LIN {X 0,Y 573.917,Z 349.97,A -85,B 0,C 180,E1 -2263.779,E2 -2263.779} C_VEL
LIN {X 0,Y 573.417,Z 346.271,A -85,B 0,C 180,E1 -2263.85,E2 -2263.85} C_VEL
LIN {X 0,Y 573.634,Z 323.251,A -85,B 0,C 180,E1 -2266.915,E2 -2266.915} C_VEL
LIN {X 0,Y 573.847,Z 301.546,A -85,B 0,C 180,E1 -2269.849,E2 -2269.849} C_VEL
LIN {X 0,Y 574.055,Z 282.107,A -85,B 0,C 180,E1 -2272.493,E2 -2272.493} C_VEL
LIN {X 0,Y 574.049,Z 273.401,A -85,B 0,C 180,E1 -2273.681,E2 -2273.681} C_VEL
LIN {X 0,Y 573.25,Z 269.082,A -85,B 0,C 180,E1 -2274.344,E2 -2274.344} C_VEL
LIN {X 0,Y 573.182,Z 269.086,A -85,B 0,C 180,E1 -2276.978,E2 -2276.978} C_VEL
LIN {X 0,Y 573.215,Z 269.077,A -85,B 0,C 180,E1 -2279.482,E2 -2279.482} C_VEL
LIN {X 0,Y 573.242,Z 269.078,A -85,B 0,C 180,E1 -2282.226,E2 -2282.226} C_VEL
LIN {X 0,Y 573.214,Z 269.085,A -85,B 0,C 180,E1 -2284.768,E2 -2284.768} C_VEL
LIN {X 0,Y 573.204,Z 269.079,A -85,B 0,C 180,E1 -2287.807,E2 -2287.807} C_VEL
LIN {X 0,Y 573.23,Z 269.083,A -85,B 0,C 180,E1 -2290.523,E2 -2290.523} C_VEL
LIN {X 0,Y 573.189,Z 269.081,A -85,B 0,C 180,E1 -2293.36,E2 -2293.36} C_VEL
LIN {X 0,Y 573.213,Z 269.082,A -85,B 0,C 180,E1 -2296.33,E2 -2296.33} C_VEL
LIN {X 0,Y 573.222,Z 269.077,A -85,B 0,C 180,E1 -2299.473,E2 -2299.473} C_VEL
LIN {X 0,Y 573.201,Z 269.082,A -85,B 0,C 180,E1 -2302.189,E2 -2302.189} C_VEL
LIN {X 0,Y 573.199,Z 269.081,A -85,B 0,C 180,E1 -2305.228,E2 -2305.228} C_VEL
LIN {X 0,Y 573.21,Z 269.08,A -85,B 0,C 180,E1 -2308.182,E2 -2308.182} C_VEL
LIN {X 0,Y 573.206,Z 269.087,A -85,B 0,C 180,E1 -2310.631,E2 -2310.631} C_VEL
LIN {X 0,Y 573.178,Z 269.087,A -85,B 0,C 180,E1 -2313.02,E2 -2313.02} C_VEL
LIN {X 0,Y 573.181,Z 269.083,A -85,B 0,C 180,E1 -2315.361,E2 -2315.361} C_VEL
LIN {X 0,Y 573.185,Z 269.081,A -85,B 0,C 180,E1 -2317.66,E2 -2317.66} C_VEL
LIN {X 0,Y 573.227,Z 269.085,A -85,B 0,C 180,E1 -2320.668,E2 -2320.668} C_VEL
LIN {X 0,Y 573.205,Z 269.079,A -85,B 0,C 180,E1 -2323.62,E2 -2323.62} C_VEL
LIN {X 0,Y 573.192,Z 269.087,A -85,B 0,C 180,E1 -2326.528,E2 -2326.528} C_VEL
LIN {X 0,Y 573.243,Z 269.075,A -85,B 0,C 180,E1 -2329.403,E2 -2329.403} C_VEL
LIN {X 0,Y 573.241,Z 269.077,A -85,B 0,C 180,E1 -2332.249,E2 -2332.249} C_VEL
LIN {X 0,Y 573.271,Z 269.076,A -85,B 0,C 180,E1 -2335.077,E2 -2335.077} C_VEL
LIN {X 0,Y 573.256,Z 269.072,A -85,B 0,C 180,E1 -2337.892,E2 -2337.892} C_VEL
LIN {X 0,Y 573.307,Z 269.075,A -85,B 0,C 180,E1 -2340.702,E2 -2340.702} C_VEL
LIN {X 0,Y 573.204,Z 269.08,A -85,B 0,C 180,E1 -2343.514,E2 -2343.514} C_VEL
LIN {X 0,Y 573.254,Z 269.073,A -85,B 0,C 180,E1 -2345.628,E2 -2345.628} C_VEL
LIN {X 0,Y 573.267,Z 269.075,A -85,B 0,C 180,E1 -2348.459,E2 -2348.459} C_VEL
LIN {X 0,Y 573.284,Z 269.072,A -85,B 0,C 180,E1 -2351.311,E2 -2351.311} C_VEL
LIN {X 0,Y 573.239,Z 269.078,A -85,B 0,C 180,E1 -2354.425,E2 -2354.425} C_VEL
LIN {X 0,Y 573.221,Z 269.083,A -85,B 0,C 180,E1 -2357.112,E2 -2357.112} C_VEL
LIN {X 0,Y 573.224,Z 269.077,A -85,B 0,C 180,E1 -2360.077,E2 -2360.077} C_VEL
LIN {X 0,Y 573.206,Z 269.081,A -85,B 0,C 180,E1 -2362.339,E2 -2362.339} C_VEL
LIN {X 0,Y 573.216,Z 269.081,A -85,B 0,C 180,E1 -2364.415,E2 -2364.415} C_VEL
LIN {X 0,Y 572.592,Z 269.165,A -85,B 0,C 180,E1 -2365.001,E2 -2365.001} C_VEL
LIN {X 0,Y 569.754,Z 269.52,A -85,B 0,C 180,E1 -2365.953,E2 -2365.953} C_VEL
LIN {X 0,Y 567.326,Z 269.819,A -85,B 0,C 180,E1 -2366.719,E2 -2366.719} C_VEL
LIN {X 0,Y 566.274,Z 269.946,A -85,B 0,C 180,E1 -2367.31,E2 -2367.31} C_VEL
LIN {X 0,Y 566.184,Z 269.955,A -85,B 0,C 180,E1 -2367.511,E2 -2367.511} C_VEL
LIN {X 0,Y 566.163,Z 269.961,A -85,B 0,C 180,E1 -2370.593,E2 -2370.593} C_VEL
LIN {X 0,Y 566.198,Z 269.959,A -85,B 0,C 180,E1 -2373.103,E2 -2373.103} C_VEL
LIN {X 0,Y 566.185,Z 269.954,A -85,B 0,C 180,E1 -2375.69,E2 -2375.69} C_VEL
LIN {X 0,Y 566.191,Z 269.957,A -85,B 0,C 180,E1 -2378.561,E2 -2378.561} C_VEL
LIN {X 0,Y 566.196,Z 269.959,A -85,B 0,C 180,E1 -2381.137,E2 -2381.137} C_VEL
LIN {X 0,Y 566.177,Z 269.954,A -85,B 0,C 180,E1 -2384.037,E2 -2384.037} C_VEL
LIN {X 0,Y 566.19,Z 269.961,A -85,B 0,C 180,E1 -2387.084,E2 -2387.084} C_VEL
LIN {X 0,Y 566.209,Z 269.951,A -85,B 0,C 180,E1 -2389.805,E2 -2389.805} C_VEL
LIN {X 0,Y 566.183,Z 269.958,A -85,B 0,C 180,E1 -2392.601,E2 -2392.601} C_VEL
LIN {X 0,Y 566.205,Z 269.958,A -85,B 0,C 180,E1 -2395.185,E2 -2395.185} C_VEL
LIN {X 0,Y 566.222,Z 269.949,A -85,B 0,C 180,E1 -2397.745,E2 -2397.745} C_VEL
LIN {X 0,Y 566.193,Z 269.954,A -85,B 0,C 180,E1 -2400.329,E2 -2400.329} C_VEL
LIN {X 0,Y 566.21,Z 269.955,A -85,B 0,C 180,E1 -2402.663,E2 -2402.663} C_VEL
LIN {X 0,Y 566.229,Z 269.957,A -85,B 0,C 180,E1 -2405.04,E2 -2405.04} C_VEL
LIN {X 0,Y 566.187,Z 269.953,A -85,B 0,C 180,E1 -2408.138,E2 -2408.138} C_VEL
LIN {X 0,Y 566.231,Z 269.951,A -85,B 0,C 180,E1 -2410.613,E2 -2410.613} C_VEL
LIN {X 0,Y 566.212,Z 269.954,A -85,B 0,C 180,E1 -2413.413,E2 -2413.413} C_VEL
LIN {X 0,Y 566.193,Z 269.953,A -85,B 0,C 180,E1 -2416.359,E2 -2416.359} C_VEL
LIN {X 0,Y 566.232,Z 269.951,A -85,B 0,C 180,E1 -2418.675,E2 -2418.675} C_VEL
LIN {X 0,Y 566.23,Z 269.952,A -85,B 0,C 180,E1 -2421.434,E2 -2421.434} C_VEL
LIN {X 0,Y 566.255,Z 269.945,A -85,B 0,C 180,E1 -2424.301,E2 -2424.301} C_VEL
LIN {X 0,Y 566.282,Z 269.941,A -85,B 0,C 180,E1 -2427.865,E2 -2427.865} C_VEL
LIN {X 0,Y 566.297,Z 269.943,A -85,B 0,C 180,E1 -2430.71,E2 -2430.71} C_VEL
LIN {X 0,Y 566.268,Z 269.949,A -85,B 0,C 180,E1 -2432.844,E2 -2432.844} C_VEL
LIN {X 0,Y 566.261,Z 269.945,A -85,B 0,C 180,E1 -2435.697,E2 -2435.697} C_VEL
LIN {X 0,Y 566.224,Z 269.95,A -85,B 0,C 180,E1 -2438.564,E2 -2438.564} C_VEL
LIN {X 0,Y 566.235,Z 269.952,A -85,B 0,C 180,E1 -2441.452,E2 -2441.452} C_VEL
LIN {X 0,Y 566.226,Z 269.949,A -85,B 0,C 180,E1 -2444.505,E2 -2444.505} C_VEL
LIN {X 0,Y 566.194,Z 269.959,A -85,B 0,C 180,E1 -2447.329,E2 -2447.329} C_VEL
LIN {X 0,Y 566.209,Z 269.95,A -85,B 0,C 180,E1 -2450.334,E2 -2450.334} C_VEL
LIN {X 0,Y 566.216,Z 269.955,A -85,B 0,C 180,E1 -2453.399,E2 -2453.399} C_VEL
LIN {X 0,Y 566.21,Z 269.952,A -85,B 0,C 180,E1 -2455.745,E2 -2455.745} C_VEL
LIN {X 0,Y 566.19,Z 269.952,A -85,B 0,C 180,E1 -2458.2,E2 -2458.2} C_VEL
LIN {X 0,Y 566.185,Z 269.961,A -85,B 0,C 180,E1 -2461.076,E2 -2461.076} C_VEL
LIN {X 0,Y 566.205,Z 269.952,A -85,B 0,C 180,E1 -2463.734,E2 -2463.734} C_VEL
LIN {X 0,Y 566.191,Z 269.953,A -85,B 0,C 180,E1 -2466.565,E2 -2466.565} C_VEL
LIN {X 0,Y 566.188,Z 269.956,A -85,B 0,C 180,E1 -2469.683,E2 -2469.683} C_VEL
LIN {X 0,Y 566.197,Z 269.953,A -85,B 0,C 180,E1 -2472.082,E2 -2472.082} C_VEL
LIN {X 0,Y 566.254,Z 270.033,A -85,B 0,C 180,E1 -2474.364,E2 -2474.364} C_VEL
LIN {X 0,Y 566.279,Z 279.677,A -85,B 0,C 180,E1 -2476.263,E2 -2476.263} C_VEL
LIN {X 0,Y 566.19,Z 288.982,A -85,B 0,C 180,E1 -2478.061,E2 -2478.061} C_VEL
LIN {X 0,Y 567.187,Z 296.049,A -85,B 0,C 180,E1 -2478.176,E2 -2478.176} C_VEL
LIN {X 0,Y 566.936,Z 395.368,A -85,B 0,C 180,E1 -2479.456,E2 -2479.456} C_VEL
LIN {X 0,Y 566.826,Z 409.344,A -85,B 0,C 180,E1 -2479.796,E2 -2479.796} C_VEL
LIN {X 0,Y 566.705,Z 421.629,A -85,B 0,C 180,E1 -2480.246,E2 -2480.246} C_VEL
LIN {X 0,Y 566.564,Z 432.139,A -85,B 0,C 180,E1 -2480.756,E2 -2480.756} C_VEL
LIN {X 0,Y 566.42,Z 442.775,A -85,B 0,C 180,E1 -2481.406,E2 -2481.406} C_VEL
LIN {X 0,Y 566.365,Z 452.067,A -85,B 0,C 180,E1 -2482.104,E2 -2482.104} C_VEL
LIN {X 0,Y 566.234,Z 460.736,A -85,B 0,C 180,E1 -2482.886,E2 -2482.886} C_VEL
LIN {X 0,Y 566.136,Z 469.017,A -85,B 0,C 180,E1 -2483.785,E2 -2483.785} C_VEL
LIN {X 0,Y 566.01,Z 477.294,A -85,B 0,C 180,E1 -2484.886,E2 -2484.886} C_VEL
LIN {X 0,Y 565.945,Z 484.05,A -85,B 0,C 180,E1 -2486.026,E2 -2486.026} C_VEL
LIN {X 0,Y 565.918,Z 488.182,A -85,B 0,C 180,E1 -2486.878,E2 -2486.878} C_VEL
LIN {X 0,Y 565.884,Z 492.888,A -85,B 0,C 180,E1 -2488.142,E2 -2488.142} C_VEL
LIN {X 0,Y 565.877,Z 496.169,A -85,B 0,C 180,E1 -2489.39,E2 -2489.39} C_VEL
LIN {X 0,Y 565.861,Z 497.855,A -85,B 0,C 180,E1 -2490.377,E2 -2490.377} C_VEL
LIN {X 0,Y 565.838,Z 498.588,A -85,B 0,C 180,E1 -2491.027,E2 -2491.027} C_VEL
LIN {X 0,Y 565.818,Z 498.965,A -85,B 0,C 180,E1 -2491.858,E2 -2491.858} C_VEL
LIN {X 0,Y 565.834,Z 498.805,A -85,B 0,C 180,E1 -2492.642,E2 -2492.642} C_VEL
LIN {X 0,Y 565.85,Z 498.2,A -85,B 0,C 180,E1 -2493.441,E2 -2493.441} C_VEL
LIN {X 0,Y 565.858,Z 497.121,A -85,B 0,C 180,E1 -2494.234,E2 -2494.234} C_VEL
LIN {X 0,Y 565.897,Z 494.476,A -85,B 0,C 180,E1 -2495.419,E2 -2495.419} C_VEL
LIN {X 0,Y 565.928,Z 490.68,A -85,B 0,C 180,E1 -2496.585,E2 -2496.585} C_VEL
LIN {X 0,Y 565.95,Z 485.642,A -85,B 0,C 180,E1 -2497.744,E2 -2497.744} C_VEL
LIN {X 0,Y 565.99,Z 480.913,A -85,B 0,C 180,E1 -2498.619,E2 -2498.619} C_VEL
LIN {X 0,Y 566.094,Z 474.044,A -85,B 0,C 180,E1 -2499.659,E2 -2499.659} C_VEL
LIN {X 0,Y 566.157,Z 466.342,A -85,B 0,C 180,E1 -2500.615,E2 -2500.615} C_VEL
LIN {X 0,Y 566.322,Z 456.139,A -85,B 0,C 180,E1 -2501.646,E2 -2501.646} C_VEL
LIN {X 0,Y 566.385,Z 445.594,A -85,B 0,C 180,E1 -2502.488,E2 -2502.488} C_VEL
LIN {X 0,Y 566.539,Z 436.194,A -85,B 0,C 180,E1 -2503.101,E2 -2503.101} C_VEL
LIN {X 0,Y 566.628,Z 426.691,A -85,B 0,C 180,E1 -2503.61,E2 -2503.61} C_VEL
LIN {X 0,Y 566.755,Z 416.899,A -85,B 0,C 180,E1 -2504.03,E2 -2504.03} C_VEL
LIN {X 0,Y 566.837,Z 406.261,A -85,B 0,C 180,E1 -2504.379,E2 -2504.379} C_VEL
LIN {X 0,Y 566.92,Z 394.133,A -85,B 0,C 180,E1 -2504.658,E2 -2504.658} C_VEL
LIN {X 0,Y 567.05,Z 293.787,A -85,B 0,C 180,E1 -2505.946,E2 -2505.946} C_VEL
LIN {X 0,Y 566.183,Z 288.859,A -85,B 0,C 180,E1 -2506.038,E2 -2506.038} C_VEL
LIN {X 0,Y 566.336,Z 273.977,A -85,B 0,C 180,E1 -2508.945,E2 -2508.945} C_VEL
LIN {X 0,Y 566.174,Z 269.958,A -85,B 0,C 180,E1 -2509.767,E2 -2509.767} C_VEL
LIN {X 0,Y 566.183,Z 269.955,A -85,B 0,C 180,E1 -2512.153,E2 -2512.153} C_VEL
LIN {X 0,Y 566.23,Z 269.957,A -85,B 0,C 180,E1 -2515.016,E2 -2515.016} C_VEL
LIN {X 0,Y 566.211,Z 269.951,A -85,B 0,C 180,E1 -2517.866,E2 -2517.866} C_VEL
LIN {X 0,Y 566.256,Z 269.951,A -85,B 0,C 180,E1 -2520.711,E2 -2520.711} C_VEL
LIN {X 0,Y 566.146,Z 269.96,A -85,B 0,C 180,E1 -2523.559,E2 -2523.559} C_VEL
LIN {X 0,Y 566.208,Z 269.951,A -85,B 0,C 180,E1 -2525.699,E2 -2525.699} C_VEL
LIN {X 0,Y 566.192,Z 269.956,A -85,B 0,C 180,E1 -2528.567,E2 -2528.567} C_VEL
LIN {X 0,Y 566.203,Z 269.954,A -85,B 0,C 180,E1 -2531.455,E2 -2531.455} C_VEL
LIN {X 0,Y 566.173,Z 269.957,A -85,B 0,C 180,E1 -2534.509,E2 -2534.509} C_VEL
LIN {X 0,Y 566.149,Z 269.962,A -85,B 0,C 180,E1 -2537.334,E2 -2537.334} C_VEL
LIN {X 0,Y 566.158,Z 269.958,A -85,B 0,C 180,E1 -2539.583,E2 -2539.583} C_VEL
LIN {X 0,Y 566.144,Z 269.958,A -85,B 0,C 180,E1 -2541.865,E2 -2541.865} C_VEL
LIN {X 0,Y 566.181,Z 269.962,A -85,B 0,C 180,E1 -2545.037,E2 -2545.037} C_VEL
LIN {X 0,Y 566.179,Z 269.96,A -85,B 0,C 180,E1 -2547.341,E2 -2547.341} C_VEL
LIN {X 0,Y 566.153,Z 269.958,A -85,B 0,C 180,E1 -2549.772,E2 -2549.772} C_VEL
LIN {X 0,Y 566.161,Z 269.956,A -85,B 0,C 180,E1 -2552.434,E2 -2552.434} C_VEL
LIN {X 0,Y 566.168,Z 269.961,A -85,B 0,C 180,E1 -2554.998,E2 -2554.998} C_VEL
LIN {X 0,Y 566.155,Z 269.962,A -85,B 0,C 180,E1 -2557.464,E2 -2557.464} C_VEL
LIN {X 0,Y 566.188,Z 269.952,A -85,B 0,C 180,E1 -2560.201,E2 -2560.201} C_VEL
LIN {X 0,Y 566.168,Z 269.961,A -85,B 0,C 180,E1 -2563.058,E2 -2563.058} C_VEL
LIN {X 0,Y 566.166,Z 269.956,A -85,B 0,C 180,E1 -2566.053,E2 -2566.053} C_VEL
LIN {X 0,Y 566.179,Z 269.957,A -85,B 0,C 180,E1 -2568.867,E2 -2568.867} C_VEL
LIN {X 0,Y 566.158,Z 269.961,A -85,B 0,C 180,E1 -2571.641,E2 -2571.641} C_VEL
LIN {X 0,Y 566.139,Z 269.959,A -85,B 0,C 180,E1 -2574.312,E2 -2574.312} C_VEL
LIN {X 0,Y 566.186,Z 269.958,A -85,B 0,C 180,E1 -2576.901,E2 -2576.901} C_VEL
LIN {X 0,Y 566.162,Z 269.967,A -85,B 0,C 180,E1 -2579.411,E2 -2579.411} C_VEL
LIN {X 0,Y 566.172,Z 269.959,A -85,B 0,C 180,E1 -2581.86,E2 -2581.86} C_VEL
LIN {X 0,Y 566.191,Z 269.955,A -85,B 0,C 180,E1 -2584.254,E2 -2584.254} C_VEL
LIN {X 0,Y 566.235,Z 270.017,A -85,B 0,C 180,E1 -2585.703,E2 -2585.703} C_VEL
LIN {X 0,Y 567.056,Z 275.86,A -85,B 0,C 180,E1 -2586.513,E2 -2586.513} C_VEL
LIN {X 0,Y 566.955,Z 296.913,A -85,B 0,C 180,E1 -2589.315,E2 -2589.315} C_VEL
LIN {X 0,Y 566.727,Z 315.073,A -85,B 0,C 180,E1 -2591.755,E2 -2591.755} C_VEL
LIN {X 0,Y 566.527,Z 334.178,A -85,B 0,C 180,E1 -2594.349,E2 -2594.349} C_VEL
LIN {X 0,Y 566.431,Z 346.452,A -85,B 0,C 180,E1 -2595.99,E2 -2595.99} C_VEL
LIN {X 0,Y 567.179,Z 352.712,A -85,B 0,C 180,E1 -2596.089,E2 -2596.089} C_VEL
LIN {X 0,Y 566.977,Z 455.07,A -85,B 0,C 180,E1 -2597.406,E2 -2597.406} C_VEL
LIN {X 0,Y 566.845,Z 467.537,A -85,B 0,C 180,E1 -2597.698,E2 -2597.698} C_VEL
LIN {X 0,Y 566.722,Z 480.435,A -85,B 0,C 180,E1 -2598.15,E2 -2598.15} C_VEL
LIN {X 0,Y 566.63,Z 492.077,A -85,B 0,C 180,E1 -2598.704,E2 -2598.704} C_VEL
LIN {X 0,Y 566.474,Z 502.939,A -85,B 0,C 180,E1 -2599.367,E2 -2599.367} C_VEL
LIN {X 0,Y 566.332,Z 513.565,A -85,B 0,C 180,E1 -2600.178,E2 -2600.178} C_VEL
LIN {X 0,Y 566.206,Z 523.133,A -85,B 0,C 180,E1 -2601.076,E2 -2601.076} C_VEL
LIN {X 0,Y 566.111,Z 530.976,A -85,B 0,C 180,E1 -2601.974,E2 -2601.974} C_VEL
LIN {X 0,Y 566,Z 538.634,A -85,B 0,C 180,E1 -2603.048,E2 -2603.048} C_VEL
LIN {X 0,Y 566.003,Z 545.688,A -85,B 0,C 180,E1 -2604.301,E2 -2604.301} C_VEL
LIN {X 0,Y 565.933,Z 550.379,A -85,B 0,C 180,E1 -2605.372,E2 -2605.372} C_VEL
LIN {X 0,Y 565.926,Z 553.962,A -85,B 0,C 180,E1 -2606.442,E2 -2606.442} C_VEL
LIN {X 0,Y 565.878,Z 555.811,A -85,B 0,C 180,E1 -2607.154,E2 -2607.154} C_VEL
LIN {X 0,Y 565.845,Z 558.186,A -85,B 0,C 180,E1 -2608.578,E2 -2608.578} C_VEL
LIN {X 0,Y 565.839,Z 559,A -85,B 0,C 180,E1 -2610.001,E2 -2610.001} C_VEL
LIN {X 0,Y 565.845,Z 558.185,A -85,B 0,C 180,E1 -2611.424,E2 -2611.424} C_VEL
LIN {X 0,Y 565.878,Z 555.808,A -85,B 0,C 180,E1 -2612.848,E2 -2612.848} C_VEL
LIN {X 0,Y 565.927,Z 552.893,A -85,B 0,C 180,E1 -2613.917,E2 -2613.917} C_VEL
LIN {X 0,Y 565.878,Z 548.946,A -85,B 0,C 180,E1 -2614.988,E2 -2614.988} C_VEL
LIN {X 0,Y 566.002,Z 543.864,A -85,B 0,C 180,E1 -2616.059,E2 -2616.059} C_VEL
LIN {X 0,Y 566.041,Z 537.465,A -85,B 0,C 180,E1 -2617.133,E2 -2617.133} C_VEL
LIN {X 0,Y 566.134,Z 529.475,A -85,B 0,C 180,E1 -2618.208,E2 -2618.208} C_VEL
LIN {X 0,Y 566.229,Z 521.333,A -85,B 0,C 180,E1 -2619.106,E2 -2619.106} C_VEL
LIN {X 0,Y 566.342,Z 511.398,A -85,B 0,C 180,E1 -2620.005,E2 -2620.005} C_VEL
LIN {X 0,Y 566.529,Z 500.301,A -85,B 0,C 180,E1 -2620.807,E2 -2620.807} C_VEL
LIN {X 0,Y 566.641,Z 489.175,A -85,B 0,C 180,E1 -2621.446,E2 -2621.446} C_VEL
LIN {X 0,Y 566.741,Z 476.983,A -85,B 0,C 180,E1 -2621.988,E2 -2621.988} C_VEL
LIN {X 0,Y 566.864,Z 464.18,A -85,B 0,C 180,E1 -2622.394,E2 -2622.394} C_VEL
LIN {X 0,Y 566.979,Z 450.61,A -85,B 0,C 180,E1 -2622.665,E2 -2622.665} C_VEL
LIN {X 0,Y 567.031,Z 350.74,A -85,B 0,C 180,E1 -2623.94,E2 -2623.94} C_VEL
LIN {X 0,Y 566.441,Z 346.271,A -85,B 0,C 180,E1 -2624.024,E2 -2624.024} C_VEL
LIN {X 0,Y 566.694,Z 322.246,A -85,B 0,C 180,E1 -2627.265,E2 -2627.265} C_VEL
LIN {X 0,Y 566.952,Z 299.903,A -85,B 0,C 180,E1 -2630.309,E2 -2630.309} C_VEL
LIN {X 0,Y 567.192,Z 279,A -85,B 0,C 180,E1 -2633.166,E2 -2633.166} C_VEL
LIN {X 0,Y 566.866,Z 273.321,A -85,B 0,C 180,E1 -2633.968,E2 -2633.968} C_VEL
LIN {X 0,Y 566.192,Z 269.962,A -85,B 0,C 180,E1 -2634.472,E2 -2634.472} C_VEL
LIN {X 0,Y 566.16,Z 269.958,A -85,B 0,C 180,E1 -2637.34,E2 -2637.34} C_VEL
LIN {X 0,Y 566.163,Z 269.956,A -85,B 0,C 180,E1 -2639.769,E2 -2639.769} C_VEL
LIN {X 0,Y 566.194,Z 269.959,A -85,B 0,C 180,E1 -2642.428,E2 -2642.428} C_VEL
LIN {X 0,Y 566.158,Z 269.96,A -85,B 0,C 180,E1 -2644.986,E2 -2644.986} C_VEL
LIN {X 0,Y 566.172,Z 269.955,A -85,B 0,C 180,E1 -2647.46,E2 -2647.46} C_VEL
LIN {X 0,Y 566.19,Z 269.955,A -85,B 0,C 180,E1 -2650.197,E2 -2650.197} C_VEL
LIN {X 0,Y 566.169,Z 269.959,A -85,B 0,C 180,E1 -2653.053,E2 -2653.053} C_VEL
LIN {X 0,Y 566.154,Z 269.958,A -85,B 0,C 180,E1 -2656.049,E2 -2656.049} C_VEL
LIN {X 0,Y 566.179,Z 269.956,A -85,B 0,C 180,E1 -2659.213,E2 -2659.213} C_VEL
LIN {X 0,Y 566.152,Z 269.957,A -85,B 0,C 180,E1 -2661.634,E2 -2661.634} C_VEL
LIN {X 0,Y 566.12,Z 269.965,A -85,B 0,C 180,E1 -2664.304,E2 -2664.304} C_VEL
LIN {X 0,Y 566.168,Z 269.962,A -85,B 0,C 180,E1 -2666.894,E2 -2666.894} C_VEL
LIN {X 0,Y 566.141,Z 269.959,A -85,B 0,C 180,E1 -2669.404,E2 -2669.404} C_VEL
LIN {X 0,Y 566.158,Z 269.957,A -85,B 0,C 180,E1 -2671.854,E2 -2671.854} C_VEL
LIN {X 0,Y 566.157,Z 269.96,A -85,B 0,C 180,E1 -2674.248,E2 -2674.248} C_VEL
LIN {X 0,Y 566.133,Z 269.961,A -85,B 0,C 180,E1 -2677.366,E2 -2677.366} C_VEL
LIN {X 0,Y 566.165,Z 269.956,A -85,B 0,C 180,E1 -2679.661,E2 -2679.661} C_VEL
LIN {X 0,Y 566.159,Z 269.965,A -85,B 0,C 180,E1 -2682.667,E2 -2682.667} C_VEL
LIN {X 0,Y 566.173,Z 269.955,A -85,B 0,C 180,E1 -2685.625,E2 -2685.625} C_VEL
LIN {X 0,Y 566.237,Z 269.955,A -85,B 0,C 180,E1 -2688.652,E2 -2688.652} C_VEL
LIN {X 0,Y 566.183,Z 269.955,A -85,B 0,C 180,E1 -2691.433,E2 -2691.433} C_VEL
LIN {X 0,Y 566.223,Z 269.951,A -85,B 0,C 180,E1 -2694.301,E2 -2694.301} C_VEL
LIN {X 0,Y 566.228,Z 269.948,A -85,B 0,C 180,E1 -2697.866,E2 -2697.866} C_VEL
LIN {X 0,Y 566.276,Z 269.95,A -85,B 0,C 180,E1 -2700.711,E2 -2700.711} C_VEL
LIN {X 0,Y 566.155,Z 269.958,A -85,B 0,C 180,E1 -2703.558,E2 -2703.558} C_VEL
LIN {X 0,Y 566.221,Z 269.949,A -85,B 0,C 180,E1 -2705.698,E2 -2705.698} C_VEL
LIN {X 0,Y 566.209,Z 269.956,A -85,B 0,C 180,E1 -2708.566,E2 -2708.566} C_VEL
LIN {X 0,Y 566.223,Z 269.95,A -85,B 0,C 180,E1 -2711.454,E2 -2711.454} C_VEL
LIN {X 0,Y 566.192,Z 269.957,A -85,B 0,C 180,E1 -2714.507,E2 -2714.507} C_VEL
LIN {X 0,Y 566.167,Z 269.959,A -85,B 0,C 180,E1 -2717.332,E2 -2717.332} C_VEL
LIN {X 0,Y 566.177,Z 269.955,A -85,B 0,C 180,E1 -2719.581,E2 -2719.581} C_VEL
LIN {X 0,Y 566.162,Z 269.956,A -85,B 0,C 180,E1 -2721.863,E2 -2721.863} C_VEL
LIN {X 0,Y 566.181,Z 269.962,A -85,B 0,C 180,E1 -2725.031,E2 -2725.031} C_VEL
LIN {X 0,Y 566.184,Z 269.955,A -85,B 0,C 180,E1 -2727.511,E2 -2727.511} C_VEL
LIN {X 0,Y 565.506,Z 270.039,A -85,B 0,C 180,E1 -2728.105,E2 -2728.105} C_VEL
LIN {X 0,Y 562.64,Z 270.402,A -85,B 0,C 180,E1 -2729.068,E2 -2729.068} C_VEL
LIN {X 0,Y 560.23,Z 270.699,A -85,B 0,C 180,E1 -2729.844,E2 -2729.844} C_VEL
LIN {X 0,Y 559.202,Z 270.827,A -85,B 0,C 180,E1 -2730.443,E2 -2730.443} C_VEL
LIN {X 0,Y 559.122,Z 270.837,A -85,B 0,C 180,E1 -2730.645,E2 -2730.645} C_VEL
LIN {X 0,Y 559.147,Z 270.831,A -85,B 0,C 180,E1 -2733.575,E2 -2733.575} C_VEL
LIN {X 0,Y 559.162,Z 270.831,A -85,B 0,C 180,E1 -2736.453,E2 -2736.453} C_VEL
LIN {X 0,Y 559.153,Z 270.838,A -85,B 0,C 180,E1 -2738.935,E2 -2738.935} C_VEL
LIN {X 0,Y 559.174,Z 270.827,A -85,B 0,C 180,E1 -2741.769,E2 -2741.769} C_VEL
LIN {X 0,Y 559.117,Z 270.841,A -85,B 0,C 180,E1 -2744.741,E2 -2744.741} C_VEL
LIN {X 0,Y 559.149,Z 270.835,A -85,B 0,C 180,E1 -2747.259,E2 -2747.259} C_VEL
LIN {X 0,Y 559.169,Z 270.828,A -85,B 0,C 180,E1 -2750.137,E2 -2750.137} C_VEL
LIN {X 0,Y 559.132,Z 270.841,A -85,B 0,C 180,E1 -2752.894,E2 -2752.894} C_VEL
LIN {X 0,Y 559.141,Z 270.833,A -85,B 0,C 180,E1 -2755.557,E2 -2755.557} C_VEL
LIN {X 0,Y 559.157,Z 270.829,A -85,B 0,C 180,E1 -2758.139,E2 -2758.139} C_VEL
LIN {X 0,Y 559.134,Z 270.836,A -85,B 0,C 180,E1 -2760.648,E2 -2760.648} C_VEL
LIN {X 0,Y 559.163,Z 270.836,A -85,B 0,C 180,E1 -2763.173,E2 -2763.173} C_VEL
LIN {X 0,Y 559.149,Z 270.833,A -85,B 0,C 180,E1 -2765.496,E2 -2765.496} C_VEL
LIN {X 0,Y 559.165,Z 270.832,A -85,B 0,C 180,E1 -2768.625,E2 -2768.625} C_VEL
LIN {X 0,Y 559.164,Z 270.837,A -85,B 0,C 180,E1 -2770.927,E2 -2770.927} C_VEL
LIN {X 0,Y 559.163,Z 270.828,A -85,B 0,C 180,E1 -2773.948,E2 -2773.948} C_VEL
LIN {X 0,Y 559.168,Z 270.828,A -85,B 0,C 180,E1 -2776.184,E2 -2776.184} C_VEL
LIN {X 0,Y 559.193,Z 270.833,A -85,B 0,C 180,E1 -2779.133,E2 -2779.133} C_VEL
LIN {X 0,Y 559.203,Z 270.823,A -85,B 0,C 180,E1 -2782.053,E2 -2782.053} C_VEL
LIN {X 0,Y 559.25,Z 270.825,A -85,B 0,C 180,E1 -2784.953,E2 -2784.953} C_VEL
LIN {X 0,Y 559.253,Z 270.817,A -85,B 0,C 180,E1 -2787.838,E2 -2787.838} C_VEL
LIN {X 0,Y 559.268,Z 270.819,A -85,B 0,C 180,E1 -2790.719,E2 -2790.719} C_VEL
LIN {X 0,Y 559.235,Z 270.825,A -85,B 0,C 180,E1 -2792.88,E2 -2792.88} C_VEL
LIN {X 0,Y 559.229,Z 270.821,A -85,B 0,C 180,E1 -2795.768,E2 -2795.768} C_VEL
LIN {X 0,Y 559.183,Z 270.829,A -85,B 0,C 180,E1 -2798.672,E2 -2798.672} C_VEL
LIN {X 0,Y 559.199,Z 270.826,A -85,B 0,C 180,E1 -2801.598,E2 -2801.598} C_VEL
LIN {X 0,Y 559.191,Z 270.826,A -85,B 0,C 180,E1 -2804.593,E2 -2804.593} C_VEL
LIN {X 0,Y 559.154,Z 270.833,A -85,B 0,C 180,E1 -2807.554,E2 -2807.554} C_VEL
LIN {X 0,Y 559.164,Z 270.829,A -85,B 0,C 180,E1 -2809.834,E2 -2809.834} C_VEL
LIN {X 0,Y 559.143,Z 270.83,A -85,B 0,C 180,E1 -2812.149,E2 -2812.149} C_VEL
LIN {X 0,Y 559.145,Z 270.831,A -85,B 0,C 180,E1 -2814.502,E2 -2814.502} C_VEL
LIN {X 0,Y 559.165,Z 270.833,A -85,B 0,C 180,E1 -2816.898,E2 -2816.898} C_VEL
LIN {X 0,Y 559.169,Z 270.828,A -85,B 0,C 180,E1 -2819.862,E2 -2819.862} C_VEL
LIN {X 0,Y 559.154,Z 270.831,A -85,B 0,C 180,E1 -2822.71,E2 -2822.71} C_VEL
LIN {X 0,Y 559.135,Z 270.839,A -85,B 0,C 180,E1 -2825.318,E2 -2825.318} C_VEL
LIN {X 0,Y 559.109,Z 270.834,A -85,B 0,C 180,E1 -2828.013,E2 -2828.013} C_VEL
LIN {X 0,Y 559.148,Z 270.834,A -85,B 0,C 180,E1 -2830.807,E2 -2830.807} C_VEL
LIN {X 0,Y 559.162,Z 270.835,A -85,B 0,C 180,E1 -2833.725,E2 -2833.725} C_VEL
LIN {X 0,Y 559.25,Z 271.036,A -85,B 0,C 180,E1 -2834.347,E2 -2834.347} C_VEL
LIN {X 0,Y 559.215,Z 282.244,A -85,B 0,C 180,E1 -2836.566,E2 -2836.566} C_VEL
LIN {X 0,Y 559.142,Z 288.907,A -85,B 0,C 180,E1 -2837.88,E2 -2837.88} C_VEL
LIN {X 0,Y 560.301,Z 296.457,A -85,B 0,C 180,E1 -2838.008,E2 -2838.008} C_VEL
LIN {X 0,Y 560.02,Z 395.757,A -85,B 0,C 180,E1 -2839.306,E2 -2839.306} C_VEL
LIN {X 0,Y 559.904,Z 409.255,A -85,B 0,C 180,E1 -2839.64,E2 -2839.64} C_VEL
LIN {X 0,Y 559.744,Z 421.917,A -85,B 0,C 180,E1 -2840.111,E2 -2840.111} C_VEL
LIN {X 0,Y 559.584,Z 432.524,A -85,B 0,C 180,E1 -2840.636,E2 -2840.636} C_VEL
LIN {X 0,Y 559.446,Z 441.889,A -85,B 0,C 180,E1 -2841.211,E2 -2841.211} C_VEL
LIN {X 0,Y 559.325,Z 450.942,A -85,B 0,C 180,E1 -2841.884,E2 -2841.884} C_VEL
LIN {X 0,Y 559.209,Z 458.95,A -85,B 0,C 180,E1 -2842.593,E2 -2842.593} C_VEL
LIN {X 0,Y 559.118,Z 467.038,A -85,B 0,C 180,E1 -2843.449,E2 -2843.449} C_VEL
LIN {X 0,Y 559.017,Z 473.256,A -85,B 0,C 180,E1 -2844.226,E2 -2844.226} C_VEL
LIN {X 0,Y 558.933,Z 479.627,A -85,B 0,C 180,E1 -2845.174,E2 -2845.174} C_VEL
LIN {X 0,Y 558.857,Z 484.722,A -85,B 0,C 180,E1 -2846.087,E2 -2846.087} C_VEL
LIN {X 0,Y 558.848,Z 488.275,A -85,B 0,C 180,E1 -2846.836,E2 -2846.836} C_VEL
LIN {X 0,Y 558.813,Z 492.949,A -85,B 0,C 180,E1 -2848.115,E2 -2848.115} C_VEL
LIN {X 0,Y 558.771,Z 495.323,A -85,B 0,C 180,E1 -2848.957,E2 -2848.957} C_VEL
LIN {X 0,Y 558.755,Z 497.653,A -85,B 0,C 180,E1 -2850.201,E2 -2850.201} C_VEL
LIN {X 0,Y 558.731,Z 498.899,A -85,B 0,C 180,E1 -2851.689,E2 -2851.689} C_VEL
LIN {X 0,Y 558.73,Z 498.588,A -85,B 0,C 180,E1 -2853.075,E2 -2853.075} C_VEL
LIN {X 0,Y 558.743,Z 497.661,A -85,B 0,C 180,E1 -2853.881,E2 -2853.881} C_VEL
LIN {X 0,Y 558.76,Z 495.832,A -85,B 0,C 180,E1 -2854.89,E2 -2854.89} C_VEL
LIN {X 0,Y 558.822,Z 493.245,A -85,B 0,C 180,E1 -2855.875,E2 -2855.875} C_VEL
LIN {X 0,Y 558.843,Z 489.063,A -85,B 0,C 180,E1 -2857.055,E2 -2857.055} C_VEL
LIN {X 0,Y 558.889,Z 483.723,A -85,B 0,C 180,E1 -2858.205,E2 -2858.205} C_VEL
LIN {X 0,Y 558.967,Z 476.663,A -85,B 0,C 180,E1 -2859.388,E2 -2859.388} C_VEL
LIN {X 0,Y 559.078,Z 469.121,A -85,B 0,C 180,E1 -2860.396,E2 -2860.396} C_VEL
LIN {X 0,Y 559.2,Z 460.847,A -85,B 0,C 180,E1 -2861.308,E2 -2861.308} C_VEL
LIN {X 0,Y 559.295,Z 452.57,A -85,B 0,C 180,E1 -2862.07,E2 -2862.07} C_VEL
LIN {X 0,Y 559.387,Z 444.539,A -85,B 0,C 180,E1 -2862.694,E2 -2862.694} C_VEL
LIN {X 0,Y 559.6,Z 435.068,A -85,B 0,C 180,E1 -2863.305,E2 -2863.305} C_VEL
LIN {X 0,Y 559.677,Z 426.249,A -85,B 0,C 180,E1 -2863.776,E2 -2863.776} C_VEL
LIN {X 0,Y 559.77,Z 416.393,A -85,B 0,C 180,E1 -2864.2,E2 -2864.2} C_VEL
LIN {X 0,Y 559.892,Z 405.519,A -85,B 0,C 180,E1 -2864.553,E2 -2864.553} C_VEL
LIN {X 0,Y 560.015,Z 393.606,A -85,B 0,C 180,E1 -2864.824,E2 -2864.824} C_VEL
LIN {X 0,Y 560.185,Z 294.859,A -85,B 0,C 180,E1 -2866.106,E2 -2866.106} C_VEL
LIN {X 0,Y 559.152,Z 288.797,A -85,B 0,C 180,E1 -2866.23,E2 -2866.23} C_VEL
LIN {X 0,Y 559.221,Z 276.702,A -85,B 0,C 180,E1 -2868.563,E2 -2868.563} C_VEL
LIN {X 0,Y 559.177,Z 270.831,A -85,B 0,C 180,E1 -2869.637,E2 -2869.637} C_VEL
LIN {X 0,Y 559.142,Z 270.84,A -85,B 0,C 180,E1 -2872.78,E2 -2872.78} C_VEL
LIN {X 0,Y 559.203,Z 270.833,A -85,B 0,C 180,E1 -2874.953,E2 -2874.953} C_VEL
LIN {X 0,Y 559.184,Z 270.826,A -85,B 0,C 180,E1 -2877.84,E2 -2877.84} C_VEL
LIN {X 0,Y 559.224,Z 270.827,A -85,B 0,C 180,E1 -2880.72,E2 -2880.72} C_VEL
LIN {X 0,Y 559.191,Z 270.833,A -85,B 0,C 180,E1 -2882.882,E2 -2882.882} C_VEL
LIN {X 0,Y 559.175,Z 270.827,A -85,B 0,C 180,E1 -2885.771,E2 -2885.771} C_VEL
LIN {X 0,Y 559.147,Z 270.835,A -85,B 0,C 180,E1 -2888.675,E2 -2888.675} C_VEL
LIN {X 0,Y 559.154,Z 270.831,A -85,B 0,C 180,E1 -2891.602,E2 -2891.602} C_VEL
LIN {X 0,Y 559.139,Z 270.834,A -85,B 0,C 180,E1 -2894.598,E2 -2894.598} C_VEL
LIN {X 0,Y 559.109,Z 270.836,A -85,B 0,C 180,E1 -2897.559,E2 -2897.559} C_VEL
LIN {X 0,Y 559.12,Z 270.833,A -85,B 0,C 180,E1 -2899.84,E2 -2899.84} C_VEL
LIN {X 0,Y 559.09,Z 270.836,A -85,B 0,C 180,E1 -2902.155,E2 -2902.155} C_VEL
LIN {X 0,Y 559.132,Z 270.838,A -85,B 0,C 180,E1 -2905.301,E2 -2905.301} C_VEL
LIN {X 0,Y 559.146,Z 270.831,A -85,B 0,C 180,E1 -2907.714,E2 -2907.714} C_VEL
LIN {X 0,Y 559.117,Z 270.841,A -85,B 0,C 180,E1 -2911.022,E2 -2911.022} C_VEL
LIN {X 0,Y 559.132,Z 270.831,A -85,B 0,C 180,E1 -2913.955,E2 -2913.955} C_VEL
LIN {X 0,Y 559.104,Z 270.844,A -85,B 0,C 180,E1 -2917.112,E2 -2917.112} C_VEL
LIN {X 0,Y 559.131,Z 270.832,A -85,B 0,C 180,E1 -2919.947,E2 -2919.947} C_VEL
LIN {X 0,Y 559.128,Z 270.834,A -85,B 0,C 180,E1 -2922.747,E2 -2922.747} C_VEL
LIN {X 0,Y 559.12,Z 270.836,A -85,B 0,C 180,E1 -2925.765,E2 -2925.765} C_VEL
LIN {X 0,Y 559.158,Z 270.828,A -85,B 0,C 180,E1 -2928.236,E2 -2928.236} C_VEL
LIN {X 0,Y 559.147,Z 270.838,A -85,B 0,C 180,E1 -2931.196,E2 -2931.196} C_VEL
LIN {X 0,Y 559.115,Z 270.838,A -85,B 0,C 180,E1 -2933.793,E2 -2933.793} C_VEL
LIN {X 0,Y 559.138,Z 270.833,A -85,B 0,C 180,E1 -2936.429,E2 -2936.429} C_VEL
LIN {X 0,Y 559.136,Z 270.838,A -85,B 0,C 180,E1 -2938.984,E2 -2938.984} C_VEL
LIN {X 0,Y 559.153,Z 270.837,A -85,B 0,C 180,E1 -2941.623,E2 -2941.623} C_VEL
LIN {X 0,Y 559.162,Z 270.832,A -85,B 0,C 180,E1 -2944.705,E2 -2944.705} C_VEL
LIN {X 0,Y 559.216,Z 270.974,A -85,B 0,C 180,E1 -2945.6,E2 -2945.6} C_VEL
LIN {X 0,Y 560.099,Z 277.032,A -85,B 0,C 180,E1 -2946.459,E2 -2946.459} C_VEL
LIN {X 0,Y 559.934,Z 299.004,A -85,B 0,C 180,E1 -2949.428,E2 -2949.428} C_VEL
LIN {X 0,Y 559.729,Z 321.817,A -85,B 0,C 180,E1 -2952.465,E2 -2952.465} C_VEL
LIN {X 0,Y 559.443,Z 343.73,A -85,B 0,C 180,E1 -2955.451,E2 -2955.451} C_VEL
LIN {X 0,Y 559.435,Z 346.452,A -85,B 0,C 180,E1 -2955.811,E2 -2955.811} C_VEL
LIN {X 0,Y 560.293,Z 353.439,A -85,B 0,C 180,E1 -2955.924,E2 -2955.924} C_VEL
LIN {X 0,Y 560.052,Z 455.069,A -85,B 0,C 180,E1 -2957.248,E2 -2957.248} C_VEL
LIN {X 0,Y 559.925,Z 467.537,A -85,B 0,C 180,E1 -2957.544,E2 -2957.544} C_VEL
LIN {X 0,Y 559.761,Z 480.437,A -85,B 0,C 180,E1 -2958.001,E2 -2958.001} C_VEL
LIN {X 0,Y 559.665,Z 491.854,A -85,B 0,C 180,E1 -2958.549,E2 -2958.549} C_VEL
LIN {X 0,Y 559.491,Z 502.937,A -85,B 0,C 180,E1 -2959.233,E2 -2959.233} C_VEL
LIN {X 0,Y 559.311,Z 513.564,A -85,B 0,C 180,E1 -2960.053,E2 -2960.053} C_VEL
LIN {X 0,Y 559.16,Z 523.133,A -85,B 0,C 180,E1 -2960.963,E2 -2960.963} C_VEL
LIN {X 0,Y 559.048,Z 530.976,A -85,B 0,C 180,E1 -2961.872,E2 -2961.872} C_VEL
LIN {X 0,Y 558.941,Z 538.634,A -85,B 0,C 180,E1 -2962.96,E2 -2962.96} C_VEL
LIN {X 0,Y 558.935,Z 545.688,A -85,B 0,C 180,E1 -2964.229,E2 -2964.229} C_VEL
LIN {X 0,Y 558.826,Z 550.379,A -85,B 0,C 180,E1 -2965.313,E2 -2965.313} C_VEL
LIN {X 0,Y 558.836,Z 553.962,A -85,B 0,C 180,E1 -2966.396,E2 -2966.396} C_VEL
LIN {X 0,Y 558.799,Z 555.811,A -85,B 0,C 180,E1 -2967.118,E2 -2967.118} C_VEL
LIN {X 0,Y 558.745,Z 558.185,A -85,B 0,C 180,E1 -2968.56,E2 -2968.56} C_VEL
LIN {X 0,Y 558.74,Z 559,A -85,B 0,C 180,E1 -2970.001,E2 -2970.001} C_VEL
LIN {X 0,Y 558.745,Z 558.184,A -85,B 0,C 180,E1 -2971.443,E2 -2971.443} C_VEL
LIN {X 0,Y 558.799,Z 555.808,A -85,B 0,C 180,E1 -2972.885,E2 -2972.885} C_VEL
LIN {X 0,Y 558.844,Z 552.893,A -85,B 0,C 180,E1 -2973.967,E2 -2973.967} C_VEL
LIN {X 0,Y 558.798,Z 548.946,A -85,B 0,C 180,E1 -2975.051,E2 -2975.051} C_VEL
LIN {X 0,Y 558.922,Z 543.864,A -85,B 0,C 180,E1 -2976.136,E2 -2976.136} C_VEL
LIN {X 0,Y 558.978,Z 537.464,A -85,B 0,C 180,E1 -2977.223,E2 -2977.223} C_VEL
LIN {X 0,Y 559.099,Z 529.475,A -85,B 0,C 180,E1 -2978.312,E2 -2978.312} C_VEL
LIN {X 0,Y 559.185,Z 521.332,A -85,B 0,C 180,E1 -2979.221,E2 -2979.221} C_VEL
LIN {X 0,Y 559.343,Z 511.397,A -85,B 0,C 180,E1 -2980.132,E2 -2980.132} C_VEL
LIN {X 0,Y 559.535,Z 500.378,A -85,B 0,C 180,E1 -2980.938,E2 -2980.938} C_VEL
LIN {X 0,Y 559.672,Z 488.459,A -85,B 0,C 180,E1 -2981.628,E2 -2981.628} C_VEL
LIN {X 0,Y 559.809,Z 475.77,A -85,B 0,C 180,E1 -2982.185,E2 -2982.185} C_VEL
LIN {X 0,Y 559.966,Z 462.35,A -85,B 0,C 180,E1 -2982.596,E2 -2982.596} C_VEL
LIN {X 0,Y 560.062,Z 449.094,A -85,B 0,C 180,E1 -2982.847,E2 -2982.847} C_VEL
LIN {X 0,Y 560.237,Z 352.132,A -85,B 0,C 180,E1 -2984.095,E2 -2984.095} C_VEL
LIN {X 0,Y 559.427,Z 346.271,A -85,B 0,C 180,E1 -2984.203,E2 -2984.203} C_VEL
LIN {X 0,Y 559.709,Z 323.839,A -85,B 0,C 180,E1 -2987.264,E2 -2987.264} C_VEL
LIN {X 0,Y 559.992,Z 300.981,A -85,B 0,C 180,E1 -2990.38,E2 -2990.38} C_VEL
LIN {X 0,Y 560.264,Z 278.681,A -85,B 0,C 180,E1 -2993.469,E2 -2993.469} C_VEL
LIN {X 0,Y 559.901,Z 274.529,A -85,B 0,C 180,E1 -2994.074,E2 -2994.074} C_VEL
LIN {X 0,Y 559.159,Z 270.838,A -85,B 0,C 180,E1 -2994.649,E2 -2994.649} C_VEL
LIN {X 0,Y 559.109,Z 270.841,A -85,B 0,C 180,E1 -2996.904,E2 -2996.904} C_VEL
LIN {X 0,Y 559.11,Z 270.835,A -85,B 0,C 180,E1 -2999.354,E2 -2999.354} C_VEL
LIN {X 0,Y 559.156,Z 270.829,A -85,B 0,C 180,E1 -3001.861,E2 -3001.861} C_VEL
LIN {X 0,Y 559.121,Z 270.84,A -85,B 0,C 180,E1 -3004.444,E2 -3004.444} C_VEL
LIN {X 0,Y 559.112,Z 270.837,A -85,B 0,C 180,E1 -3007.108,E2 -3007.108} C_VEL
LIN {X 0,Y 559.142,Z 270.831,A -85,B 0,C 180,E1 -3009.939,E2 -3009.939} C_VEL
LIN {X 0,Y 559.132,Z 270.84,A -85,B 0,C 180,E1 -3012.742,E2 -3012.742} C_VEL
LIN {X 0,Y 559.114,Z 270.834,A -85,B 0,C 180,E1 -3015.761,E2 -3015.761} C_VEL
LIN {X 0,Y 559.104,Z 270.838,A -85,B 0,C 180,E1 -3018.224,E2 -3018.224} C_VEL
LIN {X 0,Y 559.145,Z 270.832,A -85,B 0,C 180,E1 -3021.19,E2 -3021.19} C_VEL
LIN {X 0,Y 559.093,Z 270.837,A -85,B 0,C 180,E1 -3023.785,E2 -3023.785} C_VEL
LIN {X 0,Y 559.116,Z 270.839,A -85,B 0,C 180,E1 -3026.422,E2 -3026.422} C_VEL
LIN {X 0,Y 559.122,Z 270.838,A -85,B 0,C 180,E1 -3028.978,E2 -3028.978} C_VEL
LIN {X 0,Y 559.111,Z 270.834,A -85,B 0,C 180,E1 -3031.621,E2 -3031.621} C_VEL
LIN {X 0,Y 559.125,Z 270.833,A -85,B 0,C 180,E1 -3033.9,E2 -3033.9} C_VEL
LIN {X 0,Y 559.078,Z 270.843,A -85,B 0,C 180,E1 -3037.064,E2 -3037.064} C_VEL
LIN {X 0,Y 559.135,Z 270.833,A -85,B 0,C 180,E1 -3039.393,E2 -3039.393} C_VEL
LIN {X 0,Y 559.099,Z 270.836,A -85,B 0,C 180,E1 -3041.684,E2 -3041.684} C_VEL
LIN {X 0,Y 559.125,Z 270.833,A -85,B 0,C 180,E1 -3043.946,E2 -3043.946} C_VEL
LIN {X 0,Y 559.123,Z 270.835,A -85,B 0,C 180,E1 -3046.183,E2 -3046.183} C_VEL
LIN {X 0,Y 559.198,Z 270.828,A -85,B 0,C 180,E1 -3049.133,E2 -3049.133} C_VEL
LIN {X 0,Y 559.163,Z 270.829,A -85,B 0,C 180,E1 -3052.053,E2 -3052.053} C_VEL
LIN {X 0,Y 559.217,Z 270.829,A -85,B 0,C 180,E1 -3054.953,E2 -3054.953} C_VEL
LIN {X 0,Y 559.201,Z 270.823,A -85,B 0,C 180,E1 -3057.839,E2 -3057.839} C_VEL
LIN {X 0,Y 559.244,Z 270.826,A -85,B 0,C 180,E1 -3060.72,E2 -3060.72} C_VEL
LIN {X 0,Y 559.208,Z 270.832,A -85,B 0,C 180,E1 -3062.881,E2 -3062.881} C_VEL
LIN {X 0,Y 559.189,Z 270.825,A -85,B 0,C 180,E1 -3065.77,E2 -3065.77} C_VEL
LIN {X 0,Y 559.165,Z 270.836,A -85,B 0,C 180,E1 -3068.674,E2 -3068.674} C_VEL
LIN {X 0,Y 559.174,Z 270.827,A -85,B 0,C 180,E1 -3071.601,E2 -3071.601} C_VEL
LIN {X 0,Y 559.159,Z 270.835,A -85,B 0,C 180,E1 -3074.596,E2 -3074.596} C_VEL
LIN {X 0,Y 559.127,Z 270.834,A -85,B 0,C 180,E1 -3077.558,E2 -3077.558} C_VEL
LIN {X 0,Y 559.151,Z 270.836,A -85,B 0,C 180,E1 -3080.605,E2 -3080.605} C_VEL
LIN {X 0,Y 559.11,Z 270.835,A -85,B 0,C 180,E1 -3083.718,E2 -3083.718} C_VEL
LIN {X 0,Y 559.166,Z 270.828,A -85,B 0,C 180,E1 -3086.097,E2 -3086.097} C_VEL
LIN {X 0,Y 559.133,Z 270.836,A -85,B 0,C 180,E1 -3088.531,E2 -3088.531} C_VEL
LIN {X 0,Y 559.122,Z 270.837,A -85,B 0,C 180,E1 -3090.645,E2 -3090.645} C_VEL
LIN {X 0,Y 558.46,Z 270.924,A -85,B 0,C 180,E1 -3091.247,E2 -3091.247} C_VEL
LIN {X 0,Y 555.597,Z 271.28,A -85,B 0,C 180,E1 -3092.223,E2 -3092.223} C_VEL
LIN {X 0,Y 553.185,Z 271.581,A -85,B 0,C 180,E1 -3093.009,E2 -3093.009} C_VEL
LIN {X 0,Y 552.167,Z 271.701,A -85,B 0,C 180,E1 -3093.616,E2 -3093.616} C_VEL
LIN {X 0,Y 552.095,Z 271.709,A -85,B 0,C 180,E1 -3093.821,E2 -3093.821} C_VEL
LIN {X 0,Y 552.09,Z 271.717,A -85,B 0,C 180,E1 -3096.748,E2 -3096.748} C_VEL
LIN {X 0,Y 552.109,Z 271.709,A -85,B 0,C 180,E1 -3099.528,E2 -3099.528} C_VEL
LIN {X 0,Y 552.107,Z 271.71,A -85,B 0,C 180,E1 -3102.427,E2 -3102.427} C_VEL
LIN {X 0,Y 552.078,Z 271.713,A -85,B 0,C 180,E1 -3105.565,E2 -3105.565} C_VEL
LIN {X 0,Y 552.126,Z 271.711,A -85,B 0,C 180,E1 -3108.677,E2 -3108.677} C_VEL
LIN {X 0,Y 552.104,Z 271.711,A -85,B 0,C 180,E1 -3111.413,E2 -3111.413} C_VEL
LIN {X 0,Y 552.099,Z 271.709,A -85,B 0,C 180,E1 -3114.16,E2 -3114.16} C_VEL
LIN {X 0,Y 552.099,Z 271.716,A -85,B 0,C 180,E1 -3116.815,E2 -3116.815} C_VEL
LIN {X 0,Y 552.094,Z 271.713,A -85,B 0,C 180,E1 -3119.392,E2 -3119.392} C_VEL
LIN {X 0,Y 552.117,Z 271.706,A -85,B 0,C 180,E1 -3121.904,E2 -3121.904} C_VEL
LIN {X 0,Y 552.147,Z 271.707,A -85,B 0,C 180,E1 -3124.651,E2 -3124.651} C_VEL
LIN {X 0,Y 552.086,Z 271.712,A -85,B 0,C 180,E1 -3127.55,E2 -3127.55} C_VEL
LIN {X 0,Y 552.144,Z 271.704,A -85,B 0,C 180,E1 -3130.374,E2 -3130.374} C_VEL
LIN {X 0,Y 552.151,Z 271.711,A -85,B 0,C 180,E1 -3132.978,E2 -3132.978} C_VEL
LIN {X 0,Y 552.132,Z 271.704,A -85,B 0,C 180,E1 -3136.005,E2 -3136.005} C_VEL
LIN {X 0,Y 552.16,Z 271.71,A -85,B 0,C 180,E1 -3138.993,E2 -3138.993} C_VEL
LIN {X 0,Y 552.157,Z 271.701,A -85,B 0,C 180,E1 -3141.951,E2 -3141.951} C_VEL
LIN {X 0,Y 552.225,Z 271.699,A -85,B 0,C 180,E1 -3144.888,E2 -3144.888} C_VEL
LIN {X 0,Y 552.224,Z 271.693,A -85,B 0,C 180,E1 -3147.811,E2 -3147.811} C_VEL
LIN {X 0,Y 552.239,Z 271.695,A -85,B 0,C 180,E1 -3150.728,E2 -3150.728} C_VEL
LIN {X 0,Y 552.202,Z 271.702,A -85,B 0,C 180,E1 -3152.917,E2 -3152.917} C_VEL
LIN {X 0,Y 552.198,Z 271.696,A -85,B 0,C 180,E1 -3155.842,E2 -3155.842} C_VEL
LIN {X 0,Y 552.154,Z 271.706,A -85,B 0,C 180,E1 -3158.784,E2 -3158.784} C_VEL
LIN {X 0,Y 552.156,Z 271.702,A -85,B 0,C 180,E1 -3161.748,E2 -3161.748} C_VEL
LIN {X 0,Y 552.129,Z 271.708,A -85,B 0,C 180,E1 -3164.746,E2 -3164.746} C_VEL
LIN {X 0,Y 552.105,Z 271.708,A -85,B 0,C 180,E1 -3167.786,E2 -3167.786} C_VEL
LIN {X 0,Y 552.123,Z 271.705,A -85,B 0,C 180,E1 -3170.098,E2 -3170.098} C_VEL
LIN {X 0,Y 552.101,Z 271.708,A -85,B 0,C 180,E1 -3172.447,E2 -3172.447} C_VEL
LIN {X 0,Y 552.14,Z 271.709,A -85,B 0,C 180,E1 -3175.348,E2 -3175.348} C_VEL
LIN {X 0,Y 552.11,Z 271.706,A -85,B 0,C 180,E1 -3178.094,E2 -3178.094} C_VEL
LIN {X 0,Y 552.095,Z 271.71,A -85,B 0,C 180,E1 -3180.605,E2 -3180.605} C_VEL
LIN {X 0,Y 552.106,Z 271.717,A -85,B 0,C 180,E1 -3183.181,E2 -3183.181} C_VEL
LIN {X 0,Y 552.088,Z 271.71,A -85,B 0,C 180,E1 -3185.838,E2 -3185.838} C_VEL
LIN {X 0,Y 552.099,Z 271.715,A -85,B 0,C 180,E1 -3189.059,E2 -3189.059} C_VEL
LIN {X 0,Y 552.139,Z 271.711,A -85,B 0,C 180,E1 -3191.438,E2 -3191.438} C_VEL
LIN {X 0,Y 552.165,Z 271.77,A -85,B 0,C 180,E1 -3194.265,E2 -3194.265} C_VEL
LIN {X 0,Y 552.236,Z 280.86,A -85,B 0,C 180,E1 -3196.074,E2 -3196.074} C_VEL
LIN {X 0,Y 552.144,Z 289.057,A -85,B 0,C 180,E1 -3197.692,E2 -3197.692} C_VEL
LIN {X 0,Y 553.395,Z 297.217,A -85,B 0,C 180,E1 -3197.838,E2 -3197.838} C_VEL
LIN {X 0,Y 553.122,Z 395.02,A -85,B 0,C 180,E1 -3199.129,E2 -3199.129} C_VEL
LIN {X 0,Y 552.986,Z 407.989,A -85,B 0,C 180,E1 -3199.447,E2 -3199.447} C_VEL
LIN {X 0,Y 552.802,Z 421.471,A -85,B 0,C 180,E1 -3199.939,E2 -3199.939} C_VEL
LIN {X 0,Y 552.605,Z 432.909,A -85,B 0,C 180,E1 -3200.514,E2 -3200.514} C_VEL
LIN {X 0,Y 552.471,Z 441.351,A -85,B 0,C 180,E1 -3201.035,E2 -3201.035} C_VEL
LIN {X 0,Y 552.31,Z 450.268,A -85,B 0,C 180,E1 -3201.697,E2 -3201.697} C_VEL
LIN {X 0,Y 552.201,Z 458.819,A -85,B 0,C 180,E1 -3202.46,E2 -3202.46} C_VEL
LIN {X 0,Y 552.074,Z 466.799,A -85,B 0,C 180,E1 -3203.312,E2 -3203.312} C_VEL
LIN {X 0,Y 551.971,Z 473.407,A -85,B 0,C 180,E1 -3204.148,E2 -3204.148} C_VEL
LIN {X 0,Y 551.844,Z 479.313,A -85,B 0,C 180,E1 -3205.034,E2 -3205.034} C_VEL
LIN {X 0,Y 551.804,Z 484.258,A -85,B 0,C 180,E1 -3205.917,E2 -3205.917} C_VEL
LIN {X 0,Y 551.776,Z 488.361,A -85,B 0,C 180,E1 -3206.792,E2 -3206.792} C_VEL
LIN {X 0,Y 551.747,Z 491.686,A -85,B 0,C 180,E1 -3207.658,E2 -3207.658} C_VEL
LIN {X 0,Y 551.706,Z 494.463,A -85,B 0,C 180,E1 -3208.582,E2 -3208.582} C_VEL
LIN {X 0,Y 551.671,Z 497.447,A -85,B 0,C 180,E1 -3210.017,E2 -3210.017} C_VEL
LIN {X 0,Y 551.629,Z 498.617,A -85,B 0,C 180,E1 -3211.045,E2 -3211.045} C_VEL
LIN {X 0,Y 551.645,Z 498.968,A -85,B 0,C 180,E1 -3211.876,E2 -3211.876} C_VEL
LIN {X 0,Y 551.631,Z 498.588,A -85,B 0,C 180,E1 -3213.09,E2 -3213.09} C_VEL
LIN {X 0,Y 551.667,Z 497.041,A -85,B 0,C 180,E1 -3214.333,E2 -3214.333} C_VEL
LIN {X 0,Y 551.717,Z 494.355,A -85,B 0,C 180,E1 -3215.544,E2 -3215.544} C_VEL
LIN {X 0,Y 551.748,Z 490.508,A -85,B 0,C 180,E1 -3216.743,E2 -3216.743} C_VEL
LIN {X 0,Y 551.797,Z 487.333,A -85,B 0,C 180,E1 -3217.537,E2 -3217.537} C_VEL
LIN {X 0,Y 551.839,Z 481.162,A -85,B 0,C 180,E1 -3218.742,E2 -3218.742} C_VEL
LIN {X 0,Y 551.953,Z 475.129,A -85,B 0,C 180,E1 -3219.698,E2 -3219.698} C_VEL
LIN {X 0,Y 552.027,Z 469.323,A -85,B 0,C 180,E1 -3220.478,E2 -3220.478} C_VEL
LIN {X 0,Y 552.125,Z 462.577,A -85,B 0,C 180,E1 -3221.252,E2 -3221.252} C_VEL
LIN {X 0,Y 552.285,Z 453.455,A -85,B 0,C 180,E1 -3222.122,E2 -3222.122} C_VEL
LIN {X 0,Y 552.39,Z 445.322,A -85,B 0,C 180,E1 -3222.773,E2 -3222.773} C_VEL
LIN {X 0,Y 552.606,Z 436.349,A -85,B 0,C 180,E1 -3223.373,E2 -3223.373} C_VEL
LIN {X 0,Y 552.719,Z 426.81,A -85,B 0,C 180,E1 -3223.898,E2 -3223.898} C_VEL
LIN {X 0,Y 552.841,Z 417.08,A -85,B 0,C 180,E1 -3224.328,E2 -3224.328} C_VEL
LIN {X 0,Y 552.971,Z 406.753,A -85,B 0,C 180,E1 -3224.677,E2 -3224.677} C_VEL
LIN {X 0,Y 553.081,Z 394.963,A -85,B 0,C 180,E1 -3224.963,E2 -3224.963} C_VEL
LIN {X 0,Y 553.348,Z 295.929,A -85,B 0,C 180,E1 -3226.27,E2 -3226.27} C_VEL
LIN {X 0,Y 552.134,Z 288.968,A -85,B 0,C 180,E1 -3226.404,E2 -3226.404} C_VEL
LIN {X 0,Y 552.172,Z 275.63,A -85,B 0,C 180,E1 -3228.819,E2 -3228.819} C_VEL
LIN {X 0,Y 552.107,Z 271.713,A -85,B 0,C 180,E1 -3229.457,E2 -3229.457} C_VEL
LIN {X 0,Y 552.104,Z 271.709,A -85,B 0,C 180,E1 -3231.951,E2 -3231.951} C_VEL
LIN {X 0,Y 552.176,Z 271.709,A -85,B 0,C 180,E1 -3234.889,E2 -3234.889} C_VEL
LIN {X 0,Y 552.156,Z 271.702,A -85,B 0,C 180,E1 -3237.812,E2 -3237.812} C_VEL
LIN {X 0,Y 552.193,Z 271.703,A -85,B 0,C 180,E1 -3240.73,E2 -3240.73} C_VEL
LIN {X 0,Y 552.157,Z 271.71,A -85,B 0,C 180,E1 -3242.919,E2 -3242.919} C_VEL
LIN {X 0,Y 552.143,Z 271.703,A -85,B 0,C 180,E1 -3245.845,E2 -3245.845} C_VEL
LIN {X 0,Y 552.115,Z 271.712,A -85,B 0,C 180,E1 -3248.787,E2 -3248.787} C_VEL
LIN {X 0,Y 552.107,Z 271.707,A -85,B 0,C 180,E1 -3251.752,E2 -3251.752} C_VEL
LIN {X 0,Y 552.079,Z 271.716,A -85,B 0,C 180,E1 -3254.75,E2 -3254.75} C_VEL
LIN {X 0,Y 552.061,Z 271.712,A -85,B 0,C 180,E1 -3257.79,E2 -3257.79} C_VEL
LIN {X 0,Y 552.079,Z 271.709,A -85,B 0,C 180,E1 -3260.104,E2 -3260.104} C_VEL
LIN {X 0,Y 552.043,Z 271.716,A -85,B 0,C 180,E1 -3262.453,E2 -3262.453} C_VEL
LIN {X 0,Y 552.11,Z 271.711,A -85,B 0,C 180,E1 -3265.355,E2 -3265.355} C_VEL
LIN {X 0,Y 552.077,Z 271.71,A -85,B 0,C 180,E1 -3268.1,E2 -3268.1} C_VEL
LIN {X 0,Y 552.06,Z 271.715,A -85,B 0,C 180,E1 -3270.612,E2 -3270.612} C_VEL
LIN {X 0,Y 552.083,Z 271.719,A -85,B 0,C 180,E1 -3273.188,E2 -3273.188} C_VEL
LIN {X 0,Y 552.065,Z 271.713,A -85,B 0,C 180,E1 -3275.846,E2 -3275.846} C_VEL
LIN {X 0,Y 552.087,Z 271.717,A -85,B 0,C 180,E1 -3279.066,E2 -3279.066} C_VEL
LIN {X 0,Y 552.134,Z 271.709,A -85,B 0,C 180,E1 -3281.445,E2 -3281.445} C_VEL
LIN {X 0,Y 552.06,Z 271.713,A -85,B 0,C 180,E1 -3284.536,E2 -3284.536} C_VEL
LIN {X 0,Y 552.101,Z 271.713,A -85,B 0,C 180,E1 -3287.588,E2 -3287.588} C_VEL
LIN {X 0,Y 552.103,Z 271.708,A -85,B 0,C 180,E1 -3290.477,E2 -3290.477} C_VEL
LIN {X 0,Y 552.082,Z 271.72,A -85,B 0,C 180,E1 -3293.321,E2 -3293.321} C_VEL
LIN {X 0,Y 552.105,Z 271.711,A -85,B 0,C 180,E1 -3295.943,E2 -3295.943} C_VEL
LIN {X 0,Y 552.101,Z 271.711,A -85,B 0,C 180,E1 -3298.544,E2 -3298.544} C_VEL
LIN {X 0,Y 552.108,Z 271.716,A -85,B 0,C 180,E1 -3301.442,E2 -3301.442} C_VEL
LIN {X 0,Y 552.113,Z 271.709,A -85,B 0,C 180,E1 -3304.359,E2 -3304.359} C_VEL
LIN {X 0,Y 552.166,Z 271.826,A -85,B 0,C 180,E1 -3305.494,E2 -3305.494} C_VEL
LIN {X 0,Y 553.144,Z 278.866,A -85,B 0,C 180,E1 -3306.477,E2 -3306.477} C_VEL
LIN {X 0,Y 552.908,Z 301.204,A -85,B 0,C 180,E1 -3309.543,E2 -3309.543} C_VEL
LIN {X 0,Y 552.662,Z 323.088,A -85,B 0,C 180,E1 -3312.506,E2 -3312.506} C_VEL
LIN {X 0,Y 552.433,Z 345.08,A -85,B 0,C 180,E1 -3315.451,E2 -3315.451} C_VEL
LIN {X 0,Y 552.447,Z 346.442,A -85,B 0,C 180,E1 -3315.628,E2 -3315.628} C_VEL
LIN {X 0,Y 553.389,Z 354.507,A -85,B 0,C 180,E1 -3315.758,E2 -3315.758} C_VEL
LIN {X 0,Y 553.137,Z 455.069,A -85,B 0,C 180,E1 -3317.085,E2 -3317.085} C_VEL
LIN {X 0,Y 552.991,Z 467.536,A -85,B 0,C 180,E1 -3317.385,E2 -3317.385} C_VEL
LIN {X 0,Y 552.85,Z 479.976,A -85,B 0,C 180,E1 -3317.829,E2 -3317.829} C_VEL
LIN {X 0,Y 552.68,Z 491.855,A -85,B 0,C 180,E1 -3318.403,E2 -3318.403} C_VEL
LIN {X 0,Y 552.493,Z 502.935,A -85,B 0,C 180,E1 -3319.095,E2 -3319.095} C_VEL
LIN {X 0,Y 552.29,Z 513.562,A -85,B 0,C 180,E1 -3319.925,E2 -3319.925} C_VEL
LIN {X 0,Y 552.124,Z 523.133,A -85,B 0,C 180,E1 -3320.847,E2 -3320.847} C_VEL
LIN {X 0,Y 552.012,Z 530.976,A -85,B 0,C 180,E1 -3321.767,E2 -3321.767} C_VEL
LIN {X 0,Y 551.887,Z 538.633,A -85,B 0,C 180,E1 -3322.87,E2 -3322.87} C_VEL
LIN {X 0,Y 551.866,Z 545.688,A -85,B 0,C 180,E1 -3324.154,E2 -3324.154} C_VEL
LIN {X 0,Y 551.725,Z 550.379,A -85,B 0,C 180,E1 -3325.252,E2 -3325.252} C_VEL
LIN {X 0,Y 551.75,Z 553.963,A -85,B 0,C 180,E1 -3326.35,E2 -3326.35} C_VEL
LIN {X 0,Y 551.723,Z 555.81,A -85,B 0,C 180,E1 -3327.081,E2 -3327.081} C_VEL
LIN {X 0,Y 551.645,Z 558.184,A -85,B 0,C 180,E1 -3328.541,E2 -3328.541} C_VEL
LIN {X 0,Y 551.64,Z 559,A -85,B 0,C 180,E1 -3330.001,E2 -3330.001} C_VEL
LIN {X 0,Y 551.645,Z 558.183,A -85,B 0,C 180,E1 -3331.461,E2 -3331.461} C_VEL
LIN {X 0,Y 551.724,Z 555.808,A -85,B 0,C 180,E1 -3332.922,E2 -3332.922} C_VEL
LIN {X 0,Y 551.764,Z 552.893,A -85,B 0,C 180,E1 -3334.018,E2 -3334.018} C_VEL
LIN {X 0,Y 551.724,Z 548.946,A -85,B 0,C 180,E1 -3335.116,E2 -3335.116} C_VEL
LIN {X 0,Y 551.803,Z 543.189,A -85,B 0,C 180,E1 -3336.341,E2 -3336.341} C_VEL
LIN {X 0,Y 551.927,Z 536.233,A -85,B 0,C 180,E1 -3337.5,E2 -3337.5} C_VEL
LIN {X 0,Y 552.083,Z 527.989,A -85,B 0,C 180,E1 -3338.603,E2 -3338.603} C_VEL
LIN {X 0,Y 552.224,Z 519.537,A -85,B 0,C 180,E1 -3339.523,E2 -3339.523} C_VEL
LIN {X 0,Y 552.384,Z 509.091,A -85,B 0,C 180,E1 -3340.446,E2 -3340.446} C_VEL
LIN {X 0,Y 552.626,Z 498.189,A -85,B 0,C 180,E1 -3341.219,E2 -3341.219} C_VEL
LIN {X 0,Y 552.751,Z 487.405,A -85,B 0,C 180,E1 -3341.831,E2 -3341.831} C_VEL
LIN {X 0,Y 552.872,Z 475.766,A -85,B 0,C 180,E1 -3342.34,E2 -3342.34} C_VEL
LIN {X 0,Y 553.032,Z 462.349,A -85,B 0,C 180,E1 -3342.756,E2 -3342.756} C_VEL
LIN {X 0,Y 553.152,Z 449.094,A -85,B 0,C 180,E1 -3343.01,E2 -3343.01} C_VEL
LIN {X 0,Y 553.278,Z 352.084,A -85,B 0,C 180,E1 -3344.276,E2 -3344.276} C_VEL
LIN {X 0,Y 552.434,Z 346.268,A -85,B 0,C 180,E1 -3344.387,E2 -3344.387} C_VEL
LIN {X 0,Y 552.721,Z 323.361,A -85,B 0,C 180,E1 -3347.513,E2 -3347.513} C_VEL
LIN {X 0,Y 553.024,Z 300.666,A -85,B 0,C 180,E1 -3350.649,E2 -3350.649} C_VEL
LIN {X 0,Y 553.347,Z 280.118,A -85,B 0,C 180,E1 -3353.535,E2 -3353.535} C_VEL
LIN {X 0,Y 553.192,Z 277.028,A -85,B 0,C 180,E1 -3353.986,E2 -3353.986} C_VEL
LIN {X 0,Y 552.124,Z 271.713,A -85,B 0,C 180,E1 -3354.837,E2 -3354.837} C_VEL
LIN {X 0,Y 552.071,Z 271.715,A -85,B 0,C 180,E1 -3358.099,E2 -3358.099} C_VEL
LIN {X 0,Y 552.086,Z 271.719,A -85,B 0,C 180,E1 -3360.608,E2 -3360.608} C_VEL
LIN {X 0,Y 552.096,Z 271.71,A -85,B 0,C 180,E1 -3363.185,E2 -3363.185} C_VEL
LIN {X 0,Y 552.059,Z 271.713,A -85,B 0,C 180,E1 -3365.843,E2 -3365.843} C_VEL
LIN {X 0,Y 552.102,Z 271.711,A -85,B 0,C 180,E1 -3369.058,E2 -3369.058} C_VEL
LIN {X 0,Y 552.057,Z 271.713,A -85,B 0,C 180,E1 -3371.448,E2 -3371.448} C_VEL
LIN {X 0,Y 552.075,Z 271.711,A -85,B 0,C 180,E1 -3373.479,E2 -3373.479} C_VEL
LIN {X 0,Y 552.058,Z 271.721,A -85,B 0,C 180,E1 -3376.571,E2 -3376.571} C_VEL
LIN {X 0,Y 552.083,Z 271.71,A -85,B 0,C 180,E1 -3379.516,E2 -3379.516} C_VEL
LIN {X 0,Y 552.06,Z 271.717,A -85,B 0,C 180,E1 -3382.333,E2 -3382.333} C_VEL
LIN {X 0,Y 552.05,Z 271.718,A -85,B 0,C 180,E1 -3385.048,E2 -3385.048} C_VEL
LIN {X 0,Y 552.083,Z 271.71,A -85,B 0,C 180,E1 -3387.679,E2 -3387.679} C_VEL
LIN {X 0,Y 552.053,Z 271.717,A -85,B 0,C 180,E1 -3390.231,E2 -3390.231} C_VEL
LIN {X 0,Y 552.096,Z 271.714,A -85,B 0,C 180,E1 -3393,E2 -3393} C_VEL
LIN {X 0,Y 552.044,Z 271.716,A -85,B 0,C 180,E1 -3395.959,E2 -3395.959} C_VEL
LIN {X 0,Y 552.078,Z 271.715,A -85,B 0,C 180,E1 -3399.118,E2 -3399.118} C_VEL
LIN {X 0,Y 552.055,Z 271.715,A -85,B 0,C 180,E1 -3401.442,E2 -3401.442} C_VEL
LIN {X 0,Y 552.075,Z 271.711,A -85,B 0,C 180,E1 -3403.736,E2 -3403.736} C_VEL
LIN {X 0,Y 552.085,Z 271.711,A -85,B 0,C 180,E1 -3406.003,E2 -3406.003} C_VEL
LIN {X 0,Y 552.157,Z 271.707,A -85,B 0,C 180,E1 -3408.993,E2 -3408.993} C_VEL
LIN {X 0,Y 552.117,Z 271.706,A -85,B 0,C 180,E1 -3411.951,E2 -3411.951} C_VEL
LIN {X 0,Y 552.192,Z 271.705,A -85,B 0,C 180,E1 -3414.888,E2 -3414.888} C_VEL
LIN {X 0,Y 552.174,Z 271.699,A -85,B 0,C 180,E1 -3417.811,E2 -3417.811} C_VEL
LIN {X 0,Y 552.213,Z 271.702,A -85,B 0,C 180,E1 -3420.729,E2 -3420.729} C_VEL
LIN {X 0,Y 552.174,Z 271.707,A -85,B 0,C 180,E1 -3422.918,E2 -3422.918} C_VEL
LIN {X 0,Y 552.158,Z 271.701,A -85,B 0,C 180,E1 -3425.844,E2 -3425.844} C_VEL
LIN {X 0,Y 552.133,Z 271.712,A -85,B 0,C 180,E1 -3428.786,E2 -3428.786} C_VEL
LIN {X 0,Y 552.127,Z 271.705,A -85,B 0,C 180,E1 -3431.751,E2 -3431.751} C_VEL
LIN {X 0,Y 552.097,Z 271.716,A -85,B 0,C 180,E1 -3434.749,E2 -3434.749} C_VEL
LIN {X 0,Y 552.079,Z 271.711,A -85,B 0,C 180,E1 -3437.789,E2 -3437.789} C_VEL
LIN {X 0,Y 552.098,Z 271.709,A -85,B 0,C 180,E1 -3440.102,E2 -3440.102} C_VEL
LIN {X 0,Y 552.061,Z 271.717,A -85,B 0,C 180,E1 -3442.452,E2 -3442.452} C_VEL
LIN {X 0,Y 552.121,Z 271.709,A -85,B 0,C 180,E1 -3445.352,E2 -3445.352} C_VEL
LIN {X 0,Y 552.094,Z 271.71,A -85,B 0,C 180,E1 -3448.099,E2 -3448.099} C_VEL
LIN {X 0,Y 552.081,Z 271.716,A -85,B 0,C 180,E1 -3450.641,E2 -3450.641} C_VEL
LIN {X 0,Y 552.099,Z 271.714,A -85,B 0,C 180,E1 -3453.186,E2 -3453.186} C_VEL
LIN {X 0,Y 552.095,Z 271.709,A -85,B 0,C 180,E1 -3453.821,E2 -3453.821} C_VEL
LIN {X 0,Y 551.462,Z 271.792,A -85,B 0,C 180,E1 -3454.43,E2 -3454.43} C_VEL
LIN {X 0,Y 548.638,Z 272.147,A -85,B 0,C 180,E1 -3455.418,E2 -3455.418} C_VEL
LIN {X 0,Y 546.213,Z 272.452,A -85,B 0,C 180,E1 -3456.213,E2 -3456.213} C_VEL
LIN {X 0,Y 545.141,Z 272.583,A -85,B 0,C 180,E1 -3456.827,E2 -3456.827} C_VEL
LIN {X 0,Y 545.039,Z 272.594,A -85,B 0,C 180,E1 -3457.035,E2 -3457.035} C_VEL
LIN {X 0,Y 545.068,Z 272.585,A -85,B 0,C 180,E1 -3460.142,E2 -3460.142} C_VEL
LIN {X 0,Y 545.055,Z 272.593,A -85,B 0,C 180,E1 -3463.108,E2 -3463.108} C_VEL
LIN {X 0,Y 545.045,Z 272.588,A -85,B 0,C 180,E1 -3466.226,E2 -3466.226} C_VEL
LIN {X 0,Y 545.086,Z 272.59,A -85,B 0,C 180,E1 -3468.889,E2 -3468.889} C_VEL
LIN {X 0,Y 545.038,Z 272.589,A -85,B 0,C 180,E1 -3471.765,E2 -3471.765} C_VEL
LIN {X 0,Y 545.05,Z 272.59,A -85,B 0,C 180,E1 -3474.535,E2 -3474.535} C_VEL
LIN {X 0,Y 545.054,Z 272.592,A -85,B 0,C 180,E1 -3477.213,E2 -3477.213} C_VEL
LIN {X 0,Y 545.054,Z 272.586,A -85,B 0,C 180,E1 -3479.812,E2 -3479.812} C_VEL
LIN {X 0,Y 545.085,Z 272.584,A -85,B 0,C 180,E1 -3482.346,E2 -3482.346} C_VEL
LIN {X 0,Y 545.109,Z 272.586,A -85,B 0,C 180,E1 -3484.821,E2 -3484.821} C_VEL
LIN {X 0,Y 545.032,Z 272.595,A -85,B 0,C 180,E1 -3487.243,E2 -3487.243} C_VEL
LIN {X 0,Y 545.115,Z 272.58,A -85,B 0,C 180,E1 -3490.416,E2 -3490.416} C_VEL
LIN {X 0,Y 545.069,Z 272.587,A -85,B 0,C 180,E1 -3493.522,E2 -3493.522} C_VEL
LIN {X 0,Y 545.091,Z 272.582,A -85,B 0,C 180,E1 -3495.82,E2 -3495.82} C_VEL
LIN {X 0,Y 545.115,Z 272.585,A -85,B 0,C 180,E1 -3498.849,E2 -3498.849} C_VEL
LIN {X 0,Y 545.128,Z 272.577,A -85,B 0,C 180,E1 -3501.847,E2 -3501.847} C_VEL
LIN {X 0,Y 545.201,Z 272.573,A -85,B 0,C 180,E1 -3504.822,E2 -3504.822} C_VEL
LIN {X 0,Y 545.195,Z 272.569,A -85,B 0,C 180,E1 -3507.783,E2 -3507.783} C_VEL
LIN {X 0,Y 545.209,Z 272.571,A -85,B 0,C 180,E1 -3510.737,E2 -3510.737} C_VEL
LIN {X 0,Y 545.169,Z 272.579,A -85,B 0,C 180,E1 -3512.954,E2 -3512.954} C_VEL
LIN {X 0,Y 545.168,Z 272.572,A -85,B 0,C 180,E1 -3515.918,E2 -3515.918} C_VEL
LIN {X 0,Y 545.113,Z 272.585,A -85,B 0,C 180,E1 -3518.898,E2 -3518.898} C_VEL
LIN {X 0,Y 545.129,Z 272.577,A -85,B 0,C 180,E1 -3521.902,E2 -3521.902} C_VEL
LIN {X 0,Y 545.078,Z 272.589,A -85,B 0,C 180,E1 -3524.941,E2 -3524.941} C_VEL
LIN {X 0,Y 545.073,Z 272.583,A -85,B 0,C 180,E1 -3528.023,E2 -3528.023} C_VEL
LIN {X 0,Y 545.087,Z 272.582,A -85,B 0,C 180,E1 -3530.369,E2 -3530.369} C_VEL
LIN {X 0,Y 545.1,Z 272.584,A -85,B 0,C 180,E1 -3533.555,E2 -3533.555} C_VEL
LIN {X 0,Y 545.073,Z 272.583,A -85,B 0,C 180,E1 -3535.997,E2 -3535.997} C_VEL
LIN {X 0,Y 545.075,Z 272.586,A -85,B 0,C 180,E1 -3538.746,E2 -3538.746} C_VEL
LIN {X 0,Y 545.056,Z 272.588,A -85,B 0,C 180,E1 -3541.679,E2 -3541.679} C_VEL
LIN {X 0,Y 545.061,Z 272.586,A -85,B 0,C 180,E1 -3544.559,E2 -3544.559} C_VEL
LIN {X 0,Y 545.043,Z 272.596,A -85,B 0,C 180,E1 -3547.298,E2 -3547.298} C_VEL
LIN {X 0,Y 545.065,Z 272.585,A -85,B 0,C 180,E1 -3550.136,E2 -3550.136} C_VEL
LIN {X 0,Y 545.039,Z 272.591,A -85,B 0,C 180,E1 -3552.695,E2 -3552.695} C_VEL
LIN {X 0,Y 545.158,Z 272.701,A -85,B 0,C 180,E1 -3554.208,E2 -3554.208} C_VEL
LIN {X 0,Y 545.239,Z 281.126,A -85,B 0,C 180,E1 -3555.89,E2 -3555.89} C_VEL
LIN {X 0,Y 545.135,Z 289.465,A -85,B 0,C 180,E1 -3557.514,E2 -3557.514} C_VEL
LIN {X 0,Y 546.516,Z 298.187,A -85,B 0,C 180,E1 -3557.667,E2 -3557.667} C_VEL
LIN {X 0,Y 546.219,Z 395.533,A -85,B 0,C 180,E1 -3558.975,E2 -3558.975} C_VEL
LIN {X 0,Y 546.076,Z 409.153,A -85,B 0,C 180,E1 -3559.315,E2 -3559.315} C_VEL
LIN {X 0,Y 545.85,Z 422.646,A -85,B 0,C 180,E1 -3559.829,E2 -3559.829} C_VEL
LIN {X 0,Y 545.63,Z 433.656,A -85,B 0,C 180,E1 -3560.398,E2 -3560.398} C_VEL
LIN {X 0,Y 545.48,Z 442.628,A -85,B 0,C 180,E1 -3560.972,E2 -3560.972} C_VEL
LIN {X 0,Y 545.318,Z 451.625,A -85,B 0,C 180,E1 -3561.668,E2 -3561.668} C_VEL
LIN {X 0,Y 545.189,Z 459.166,A -85,B 0,C 180,E1 -3562.36,E2 -3562.36} C_VEL
LIN {X 0,Y 545.042,Z 467.058,A -85,B 0,C 180,E1 -3563.222,E2 -3563.222} C_VEL
LIN {X 0,Y 544.926,Z 473.168,A -85,B 0,C 180,E1 -3564.008,E2 -3564.008} C_VEL
LIN {X 0,Y 544.774,Z 479.433,A -85,B 0,C 180,E1 -3564.965,E2 -3564.965} C_VEL
LIN {X 0,Y 544.724,Z 484.911,A -85,B 0,C 180,E1 -3565.976,E2 -3565.976} C_VEL
LIN {X 0,Y 544.664,Z 489.387,A -85,B 0,C 180,E1 -3566.994,E2 -3566.994} C_VEL
LIN {X 0,Y 544.64,Z 493.066,A -85,B 0,C 180,E1 -3568.058,E2 -3568.058} C_VEL
LIN {X 0,Y 544.58,Z 495.399,A -85,B 0,C 180,E1 -3568.922,E2 -3568.922} C_VEL
LIN {X 0,Y 544.589,Z 497.219,A -85,B 0,C 180,E1 -3569.83,E2 -3569.83} C_VEL
LIN {X 0,Y 544.558,Z 498.744,A -85,B 0,C 180,E1 -3571.341,E2 -3571.341} C_VEL
LIN {X 0,Y 544.549,Z 498.919,A -85,B 0,C 180,E1 -3572.315,E2 -3572.315} C_VEL
LIN {X 0,Y 544.537,Z 498.56,A -85,B 0,C 180,E1 -3573.146,E2 -3573.146} C_VEL
LIN {X 0,Y 544.592,Z 496.583,A -85,B 0,C 180,E1 -3574.588,E2 -3574.588} C_VEL
LIN {X 0,Y 544.658,Z 493.105,A -85,B 0,C 180,E1 -3576.017,E2 -3576.017} C_VEL
LIN {X 0,Y 544.668,Z 490.421,A -85,B 0,C 180,E1 -3576.825,E2 -3576.825} C_VEL
LIN {X 0,Y 544.723,Z 487.226,A -85,B 0,C 180,E1 -3577.629,E2 -3577.629} C_VEL
LIN {X 0,Y 544.755,Z 481.181,A -85,B 0,C 180,E1 -3578.824,E2 -3578.824} C_VEL
LIN {X 0,Y 544.892,Z 475.079,A -85,B 0,C 180,E1 -3579.806,E2 -3579.806} C_VEL
LIN {X 0,Y 544.985,Z 469.23,A -85,B 0,C 180,E1 -3580.606,E2 -3580.606} C_VEL
LIN {X 0,Y 545.12,Z 462.48,A -85,B 0,C 180,E1 -3581.392,E2 -3581.392} C_VEL
LIN {X 0,Y 545.265,Z 455.018,A -85,B 0,C 180,E1 -3582.131,E2 -3582.131} C_VEL
LIN {X 0,Y 545.405,Z 446.27,A -85,B 0,C 180,E1 -3582.857,E2 -3582.857} C_VEL
LIN {X 0,Y 545.642,Z 436.222,A -85,B 0,C 180,E1 -3583.539,E2 -3583.539} C_VEL
LIN {X 0,Y 545.774,Z 426.609,A -85,B 0,C 180,E1 -3584.072,E2 -3584.072} C_VEL
LIN {X 0,Y 545.915,Z 417.034,A -85,B 0,C 180,E1 -3584.495,E2 -3584.495} C_VEL
LIN {X 0,Y 546.04,Z 406.122,A -85,B 0,C 180,E1 -3584.862,E2 -3584.862} C_VEL
LIN {X 0,Y 546.161,Z 394.579,A -85,B 0,C 180,E1 -3585.135,E2 -3585.135} C_VEL
LIN {X 0,Y 546.434,Z 296.521,A -85,B 0,C 180,E1 -3586.449,E2 -3586.449} C_VEL
LIN {X 0,Y 545.109,Z 289.003,A -85,B 0,C 180,E1 -3586.605,E2 -3586.605} C_VEL
LIN {X 0,Y 545.088,Z 284.624,A -85,B 0,C 180,E1 -3587.339,E2 -3587.339} C_VEL
LIN {X 0,Y 545.066,Z 280.441,A -85,B 0,C 180,E1 -3588.095,E2 -3588.095} C_VEL
LIN {X 0,Y 545.053,Z 272.593,A -85,B 0,C 180,E1 -3589.413,E2 -3589.413} C_VEL
LIN {X 0,Y 545.074,Z 272.585,A -85,B 0,C 180,E1 -3591.847,E2 -3591.847} C_VEL
LIN {X 0,Y 545.151,Z 272.583,A -85,B 0,C 180,E1 -3594.823,E2 -3594.823} C_VEL
LIN {X 0,Y 545.129,Z 272.578,A -85,B 0,C 180,E1 -3597.784,E2 -3597.784} C_VEL
LIN {X 0,Y 545.162,Z 272.579,A -85,B 0,C 180,E1 -3600.739,E2 -3600.739} C_VEL
LIN {X 0,Y 545.123,Z 272.586,A -85,B 0,C 180,E1 -3602.956,E2 -3602.956} C_VEL
LIN {X 0,Y 545.113,Z 272.578,A -85,B 0,C 180,E1 -3605.92,E2 -3605.92} C_VEL
LIN {X 0,Y 545.073,Z 272.591,A -85,B 0,C 180,E1 -3608.901,E2 -3608.901} C_VEL
LIN {X 0,Y 545.078,Z 272.583,A -85,B 0,C 180,E1 -3611.906,E2 -3611.906} C_VEL
LIN {X 0,Y 545.049,Z 272.595,A -85,B 0,C 180,E1 -3614.945,E2 -3614.945} C_VEL
LIN {X 0,Y 545.031,Z 272.587,A -85,B 0,C 180,E1 -3618.028,E2 -3618.028} C_VEL
LIN {X 0,Y 545.044,Z 272.586,A -85,B 0,C 180,E1 -3620.374,E2 -3620.374} C_VEL
LIN {X 0,Y 545.037,Z 272.59,A -85,B 0,C 180,E1 -3623.562,E2 -3623.562} C_VEL
LIN {X 0,Y 545.04,Z 272.586,A -85,B 0,C 180,E1 -3626.003,E2 -3626.003} C_VEL
LIN {X 0,Y 545.041,Z 272.591,A -85,B 0,C 180,E1 -3628.752,E2 -3628.752} C_VEL
LIN {X 0,Y 545.031,Z 272.59,A -85,B 0,C 180,E1 -3631.686,E2 -3631.686} C_VEL
LIN {X 0,Y 545.04,Z 272.588,A -85,B 0,C 180,E1 -3634.566,E2 -3634.566} C_VEL
LIN {X 0,Y 544.998,Z 272.6,A -85,B 0,C 180,E1 -3637.307,E2 -3637.307} C_VEL
LIN {X 0,Y 545.055,Z 272.585,A -85,B 0,C 180,E1 -3640.144,E2 -3640.144} C_VEL
LIN {X 0,Y 545.028,Z 272.59,A -85,B 0,C 180,E1 -3642.701,E2 -3642.701} C_VEL
LIN {X 0,Y 545.026,Z 272.591,A -85,B 0,C 180,E1 -3645.875,E2 -3645.875} C_VEL
LIN {X 0,Y 545.067,Z 272.588,A -85,B 0,C 180,E1 -3648.891,E2 -3648.891} C_VEL
LIN {X 0,Y 545.025,Z 272.592,A -85,B 0,C 180,E1 -3651.766,E2 -3651.766} C_VEL
LIN {X 0,Y 545.014,Z 272.592,A -85,B 0,C 180,E1 -3654.535,E2 -3654.535} C_VEL
LIN {X 0,Y 545.047,Z 272.597,A -85,B 0,C 180,E1 -3657.215,E2 -3657.215} C_VEL
LIN {X 0,Y 545.045,Z 272.592,A -85,B 0,C 180,E1 -3659.814,E2 -3659.814} C_VEL
LIN {X 0,Y 545.044,Z 272.589,A -85,B 0,C 180,E1 -3662.346,E2 -3662.346} C_VEL
LIN {X 0,Y 545.143,Z 272.678,A -85,B 0,C 180,E1 -3665.386,E2 -3665.386} C_VEL
LIN {X 0,Y 546.11,Z 278.98,A -85,B 0,C 180,E1 -3666.28,E2 -3666.28} C_VEL
LIN {X 0,Y 545.969,Z 297.812,A -85,B 0,C 180,E1 -3668.877,E2 -3668.877} C_VEL
LIN {X 0,Y 545.662,Z 320.513,A -85,B 0,C 180,E1 -3671.997,E2 -3671.997} C_VEL
LIN {X 0,Y 545.397,Z 341.684,A -85,B 0,C 180,E1 -3674.877,E2 -3674.877} C_VEL
LIN {X 0,Y 545.376,Z 345.748,A -85,B 0,C 180,E1 -3675.427,E2 -3675.427} C_VEL
LIN {X 0,Y 546.498,Z 354.512,A -85,B 0,C 180,E1 -3675.585,E2 -3675.585} C_VEL
LIN {X 0,Y 546.216,Z 454.66,A -85,B 0,C 180,E1 -3676.919,E2 -3676.919} C_VEL
LIN {X 0,Y 546.041,Z 468.023,A -85,B 0,C 180,E1 -3677.246,E2 -3677.246} C_VEL
LIN {X 0,Y 545.888,Z 480.262,A -85,B 0,C 180,E1 -3677.691,E2 -3677.691} C_VEL
LIN {X 0,Y 545.691,Z 492.621,A -85,B 0,C 180,E1 -3678.3,E2 -3678.3} C_VEL
LIN {X 0,Y 545.499,Z 504.224,A -85,B 0,C 180,E1 -3679.048,E2 -3679.048} C_VEL
LIN {X 0,Y 545.261,Z 514.63,A -85,B 0,C 180,E1 -3679.888,E2 -3679.888} C_VEL
LIN {X 0,Y 545.083,Z 523.134,A -85,B 0,C 180,E1 -3680.727,E2 -3680.727} C_VEL
LIN {X 0,Y 544.976,Z 530.976,A -85,B 0,C 180,E1 -3681.66,E2 -3681.66} C_VEL
LIN {X 0,Y 544.822,Z 538.633,A -85,B 0,C 180,E1 -3682.777,E2 -3682.777} C_VEL
LIN {X 0,Y 544.775,Z 545.688,A -85,B 0,C 180,E1 -3684.078,E2 -3684.078} C_VEL
LIN {X 0,Y 544.628,Z 550.379,A -85,B 0,C 180,E1 -3685.19,E2 -3685.19} C_VEL
LIN {X 0,Y 544.669,Z 553.962,A -85,B 0,C 180,E1 -3686.302,E2 -3686.302} C_VEL
LIN {X 0,Y 544.65,Z 555.81,A -85,B 0,C 180,E1 -3687.043,E2 -3687.043} C_VEL
LIN {X 0,Y 544.546,Z 558.184,A -85,B 0,C 180,E1 -3688.522,E2 -3688.522} C_VEL
LIN {X 0,Y 544.541,Z 559,A -85,B 0,C 180,E1 -3690.001,E2 -3690.001} C_VEL
LIN {X 0,Y 544.546,Z 558.183,A -85,B 0,C 180,E1 -3691.48,E2 -3691.48} C_VEL
LIN {X 0,Y 544.651,Z 555.808,A -85,B 0,C 180,E1 -3692.96,E2 -3692.96} C_VEL
LIN {X 0,Y 544.684,Z 552.893,A -85,B 0,C 180,E1 -3694.07,E2 -3694.07} C_VEL
LIN {X 0,Y 544.654,Z 548.945,A -85,B 0,C 180,E1 -3695.183,E2 -3695.183} C_VEL
LIN {X 0,Y 544.74,Z 543.704,A -85,B 0,C 180,E1 -3696.328,E2 -3696.328} C_VEL
LIN {X 0,Y 544.837,Z 537.463,A -85,B 0,C 180,E1 -3697.412,E2 -3697.412} C_VEL
LIN {X 0,Y 545.007,Z 529.474,A -85,B 0,C 180,E1 -3698.528,E2 -3698.528} C_VEL
LIN {X 0,Y 545.154,Z 521.33,A -85,B 0,C 180,E1 -3699.461,E2 -3699.461} C_VEL
LIN {X 0,Y 545.341,Z 511.395,A -85,B 0,C 180,E1 -3700.395,E2 -3700.395} C_VEL
LIN {X 0,Y 545.583,Z 500.542,A -85,B 0,C 180,E1 -3701.21,E2 -3701.21} C_VEL
LIN {X 0,Y 545.741,Z 489.092,A -85,B 0,C 180,E1 -3701.891,E2 -3701.891} C_VEL
LIN {X 0,Y 545.898,Z 476.804,A -85,B 0,C 180,E1 -3702.453,E2 -3702.453} C_VEL
LIN {X 0,Y 546.112,Z 463.899,A -85,B 0,C 180,E1 -3702.873,E2 -3702.873} C_VEL
LIN {X 0,Y 546.213,Z 450.181,A -85,B 0,C 180,E1 -3703.155,E2 -3703.155} C_VEL
LIN {X 0,Y 546.422,Z 353.08,A -85,B 0,C 180,E1 -3704.437,E2 -3704.437} C_VEL
LIN {X 0,Y 545.431,Z 346.084,A -85,B 0,C 180,E1 -3704.56,E2 -3704.56} C_VEL
LIN {X 0,Y 545.723,Z 322.946,A -85,B 0,C 180,E1 -3707.759,E2 -3707.759} C_VEL
LIN {X 0,Y 546.112,Z 298.96,A -85,B 0,C 180,E1 -3711.12,E2 -3711.12} C_VEL
LIN {X 0,Y 546.422,Z 280.493,A -85,B 0,C 180,E1 -3713.758,E2 -3713.758} C_VEL
LIN {X 0,Y 545.63,Z 275.358,A -85,B 0,C 180,E1 -3714.543,E2 -3714.543} C_VEL
LIN {X 0,Y 545.074,Z 272.591,A -85,B 0,C 180,E1 -3714.976,E2 -3714.976} C_VEL
LIN {X 0,Y 545.037,Z 272.589,A -85,B 0,C 180,E1 -3717.657,E2 -3717.657} C_VEL
LIN {X 0,Y 545.037,Z 272.592,A -85,B 0,C 180,E1 -3720.238,E2 -3720.238} C_VEL
LIN {X 0,Y 545.064,Z 272.587,A -85,B 0,C 180,E1 -3723.059,E2 -3723.059} C_VEL
LIN {X 0,Y 545.01,Z 272.591,A -85,B 0,C 180,E1 -3725.669,E2 -3725.669} C_VEL
LIN {X 0,Y 545.03,Z 272.592,A -85,B 0,C 180,E1 -3728.236,E2 -3728.236} C_VEL
LIN {X 0,Y 545.011,Z 272.594,A -85,B 0,C 180,E1 -3731.118,E2 -3731.118} C_VEL
LIN {X 0,Y 545.02,Z 272.592,A -85,B 0,C 180,E1 -3734.129,E2 -3734.129} C_VEL
LIN {X 0,Y 545.006,Z 272.598,A -85,B 0,C 180,E1 -3736.886,E2 -3736.886} C_VEL
LIN {X 0,Y 545.039,Z 272.588,A -85,B 0,C 180,E1 -3739.855,E2 -3739.855} C_VEL
LIN {X 0,Y 545.039,Z 272.591,A -85,B 0,C 180,E1 -3743.073,E2 -3743.073} C_VEL
LIN {X 0,Y 545.018,Z 272.594,A -85,B 0,C 180,E1 -3746.324,E2 -3746.324} C_VEL
LIN {X 0,Y 545.033,Z 272.594,A -85,B 0,C 180,E1 -3748.95,E2 -3748.95} C_VEL
LIN {X 0,Y 545.048,Z 272.587,A -85,B 0,C 180,E1 -3751.504,E2 -3751.504} C_VEL
LIN {X 0,Y 545.018,Z 272.591,A -85,B 0,C 180,E1 -3753.996,E2 -3753.996} C_VEL
LIN {X 0,Y 544.994,Z 272.596,A -85,B 0,C 180,E1 -3757.24,E2 -3757.24} C_VEL
LIN {X 0,Y 545.078,Z 272.588,A -85,B 0,C 180,E1 -3760.413,E2 -3760.413} C_VEL
LIN {X 0,Y 545.025,Z 272.59,A -85,B 0,C 180,E1 -3763.519,E2 -3763.519} C_VEL
LIN {X 0,Y 545.046,Z 272.587,A -85,B 0,C 180,E1 -3765.818,E2 -3765.818} C_VEL
LIN {X 0,Y 545.107,Z 272.588,A -85,B 0,C 180,E1 -3768.849,E2 -3768.849} C_VEL
LIN {X 0,Y 545.087,Z 272.582,A -85,B 0,C 180,E1 -3771.846,E2 -3771.846} C_VEL
LIN {X 0,Y 545.167,Z 272.58,A -85,B 0,C 180,E1 -3774.822,E2 -3774.822} C_VEL
LIN {X 0,Y 545.147,Z 272.574,A -85,B 0,C 180,E1 -3777.783,E2 -3777.783} C_VEL
LIN {X 0,Y 545.181,Z 272.578,A -85,B 0,C 180,E1 -3780.738,E2 -3780.738} C_VEL
LIN {X 0,Y 545.14,Z 272.583,A -85,B 0,C 180,E1 -3782.956,E2 -3782.956} C_VEL
LIN {X 0,Y 545.129,Z 272.577,A -85,B 0,C 180,E1 -3785.92,E2 -3785.92} C_VEL
LIN {X 0,Y 545.09,Z 272.59,A -85,B 0,C 180,E1 -3788.9,E2 -3788.9} C_VEL
LIN {X 0,Y 545.098,Z 272.581,A -85,B 0,C 180,E1 -3791.905,E2 -3791.905} C_VEL
LIN {X 0,Y 545.047,Z 272.595,A -85,B 0,C 180,E1 -3794.944,E2 -3794.944} C_VEL
LIN {X 0,Y 545.048,Z 272.587,A -85,B 0,C 180,E1 -3798.026,E2 -3798.026} C_VEL
LIN {X 0,Y 545.063,Z 272.588,A -85,B 0,C 180,E1 -3800.373,E2 -3800.373} C_VEL
LIN {X 0,Y 545.055,Z 272.587,A -85,B 0,C 180,E1 -3803.56,E2 -3803.56} C_VEL
LIN {X 0,Y 545.055,Z 272.586,A -85,B 0,C 180,E1 -3806.001,E2 -3806.001} C_VEL
LIN {X 0,Y 545.06,Z 272.593,A -85,B 0,C 180,E1 -3808.751,E2 -3808.751} C_VEL
LIN {X 0,Y 545.047,Z 272.588,A -85,B 0,C 180,E1 -3811.684,E2 -3811.684} C_VEL
LIN {X 0,Y 545.056,Z 272.59,A -85,B 0,C 180,E1 -3814.564,E2 -3814.564} C_VEL
LIN {X 0,Y 545.039,Z 272.594,A -85,B 0,C 180,E1 -3817.035,E2 -3817.035} C_VEL
LIN {X 0,Y 544.333,Z 272.68,A -85,B 0,C 180,E1 -3817.651,E2 -3817.651} C_VEL
LIN {X 0,Y 541.479,Z 273.037,A -85,B 0,C 180,E1 -3818.652,E2 -3818.652} C_VEL
LIN {X 0,Y 539.102,Z 273.33,A -85,B 0,C 180,E1 -3819.458,E2 -3819.458} C_VEL
LIN {X 0,Y 538.098,Z 273.453,A -85,B 0,C 180,E1 -3820.08,E2 -3820.08} C_VEL
LIN {X 0,Y 538.024,Z 273.463,A -85,B 0,C 180,E1 -3820.291,E2 -3820.291} C_VEL
LIN {X 0,Y 538.003,Z 273.472,A -85,B 0,C 180,E1 -3822.989,E2 -3822.989} C_VEL
LIN {X 0,Y 538.009,Z 273.464,A -85,B 0,C 180,E1 -3825.927,E2 -3825.927} C_VEL
LIN {X 0,Y 538.061,Z 273.463,A -85,B 0,C 180,E1 -3829.251,E2 -3829.251} C_VEL
LIN {X 0,Y 537.986,Z 273.467,A -85,B 0,C 180,E1 -3832.125,E2 -3832.125} C_VEL
LIN {X 0,Y 538.005,Z 273.472,A -85,B 0,C 180,E1 -3834.919,E2 -3834.919} C_VEL
LIN {X 0,Y 538.005,Z 273.466,A -85,B 0,C 180,E1 -3837.619,E2 -3837.619} C_VEL
LIN {X 0,Y 538.007,Z 273.465,A -85,B 0,C 180,E1 -3840.24,E2 -3840.24} C_VEL
LIN {X 0,Y 538.058,Z 273.464,A -85,B 0,C 180,E1 -3842.797,E2 -3842.797} C_VEL
LIN {X 0,Y 538.04,Z 273.465,A -85,B 0,C 180,E1 -3845.294,E2 -3845.294} C_VEL
LIN {X 0,Y 538.017,Z 273.466,A -85,B 0,C 180,E1 -3848.547,E2 -3848.547} C_VEL
LIN {X 0,Y 538.033,Z 273.469,A -85,B 0,C 180,E1 -3850.941,E2 -3850.941} C_VEL
LIN {X 0,Y 538.021,Z 273.468,A -85,B 0,C 180,E1 -3853.299,E2 -3853.299} C_VEL
LIN {X 0,Y 538.06,Z 273.459,A -85,B 0,C 180,E1 -3855.631,E2 -3855.631} C_VEL
LIN {X 0,Y 538.075,Z 273.46,A -85,B 0,C 180,E1 -3858.701,E2 -3858.701} C_VEL
LIN {X 0,Y 538.085,Z 273.455,A -85,B 0,C 180,E1 -3861.739,E2 -3861.739} C_VEL
LIN {X 0,Y 538.158,Z 273.45,A -85,B 0,C 180,E1 -3864.754,E2 -3864.754} C_VEL
LIN {X 0,Y 538.167,Z 273.445,A -85,B 0,C 180,E1 -3867.754,E2 -3867.754} C_VEL
LIN {X 0,Y 538.179,Z 273.447,A -85,B 0,C 180,E1 -3870.747,E2 -3870.747} C_VEL
LIN {X 0,Y 538.136,Z 273.456,A -85,B 0,C 180,E1 -3872.993,E2 -3872.993} C_VEL
LIN {X 0,Y 538.117,Z 273.45,A -85,B 0,C 180,E1 -3875.996,E2 -3875.996} C_VEL
LIN {X 0,Y 538.064,Z 273.465,A -85,B 0,C 180,E1 -3879.016,E2 -3879.016} C_VEL
LIN {X 0,Y 538.077,Z 273.455,A -85,B 0,C 180,E1 -3882.06,E2 -3882.06} C_VEL
LIN {X 0,Y 538.038,Z 273.468,A -85,B 0,C 180,E1 -3885.141,E2 -3885.141} C_VEL
LIN {X 0,Y 538.025,Z 273.461,A -85,B 0,C 180,E1 -3888.267,E2 -3888.267} C_VEL
LIN {X 0,Y 538.031,Z 273.463,A -85,B 0,C 180,E1 -3890.648,E2 -3890.648} C_VEL
LIN {X 0,Y 538.026,Z 273.462,A -85,B 0,C 180,E1 -3893.883,E2 -3893.883} C_VEL
LIN {X 0,Y 538.034,Z 273.46,A -85,B 0,C 180,E1 -3896.363,E2 -3896.363} C_VEL
LIN {X 0,Y 538.036,Z 273.465,A -85,B 0,C 180,E1 -3898.935,E2 -3898.935} C_VEL
LIN {X 0,Y 538.006,Z 273.464,A -85,B 0,C 180,E1 -3901.887,E2 -3901.887} C_VEL
LIN {X 0,Y 538.01,Z 273.464,A -85,B 0,C 180,E1 -3904.618,E2 -3904.618} C_VEL
LIN {X 0,Y 537.999,Z 273.473,A -85,B 0,C 180,E1 -3907.17,E2 -3907.17} C_VEL
LIN {X 0,Y 538.028,Z 273.464,A -85,B 0,C 180,E1 -3909.79,E2 -3909.79} C_VEL
LIN {X 0,Y 538.035,Z 273.468,A -85,B 0,C 180,E1 -3912.989,E2 -3912.989} C_VEL
LIN {X 0,Y 538.123,Z 273.628,A -85,B 0,C 180,E1 -3914.145,E2 -3914.145} C_VEL
LIN {X 0,Y 538.243,Z 279.734,A -85,B 0,C 180,E1 -3915.365,E2 -3915.365} C_VEL
LIN {X 0,Y 538.156,Z 289.593,A -85,B 0,C 180,E1 -3917.318,E2 -3917.318} C_VEL
LIN {X 0,Y 539.658,Z 298.657,A -85,B 0,C 180,E1 -3917.486,E2 -3917.486} C_VEL
LIN {X 0,Y 539.275,Z 396.229,A -85,B 0,C 180,E1 -3918.819,E2 -3918.819} C_VEL
LIN {X 0,Y 539.167,Z 409.829,A -85,B 0,C 180,E1 -3919.168,E2 -3919.168} C_VEL
LIN {X 0,Y 538.928,Z 422.924,A -85,B 0,C 180,E1 -3919.674,E2 -3919.674} C_VEL
LIN {X 0,Y 538.686,Z 434.177,A -85,B 0,C 180,E1 -3920.262,E2 -3920.262} C_VEL
LIN {X 0,Y 538.501,Z 443.235,A -85,B 0,C 180,E1 -3920.851,E2 -3920.851} C_VEL
LIN {X 0,Y 538.321,Z 452.212,A -85,B 0,C 180,E1 -3921.557,E2 -3921.557} C_VEL
LIN {X 0,Y 538.164,Z 460.375,A -85,B 0,C 180,E1 -3922.325,E2 -3922.325} C_VEL
LIN {X 0,Y 538.009,Z 467.077,A -85,B 0,C 180,E1 -3923.066,E2 -3923.066} C_VEL
LIN {X 0,Y 537.856,Z 474.863,A -85,B 0,C 180,E1 -3924.099,E2 -3924.099} C_VEL
LIN {X 0,Y 537.738,Z 479.917,A -85,B 0,C 180,E1 -3924.897,E2 -3924.897} C_VEL
LIN {X 0,Y 537.66,Z 484.772,A -85,B 0,C 180,E1 -3925.801,E2 -3925.801} C_VEL
LIN {X 0,Y 537.616,Z 489.086,A -85,B 0,C 180,E1 -3926.776,E2 -3926.776} C_VEL
LIN {X 0,Y 537.59,Z 492.071,A -85,B 0,C 180,E1 -3927.589,E2 -3927.589} C_VEL
LIN {X 0,Y 537.54,Z 494.604,A -85,B 0,C 180,E1 -3928.468,E2 -3928.468} C_VEL
LIN {X 0,Y 537.493,Z 497.12,A -85,B 0,C 180,E1 -3929.641,E2 -3929.641} C_VEL
LIN {X 0,Y 537.454,Z 498.852,A -85,B 0,C 180,E1 -3931.165,E2 -3931.165} C_VEL
LIN {X 0,Y 537.442,Z 499.147,A -85,B 0,C 180,E1 -3931.917,E2 -3931.917} C_VEL
LIN {X 0,Y 537.438,Z 498.918,A -85,B 0,C 180,E1 -3932.762,E2 -3932.762} C_VEL
LIN {X 0,Y 537.462,Z 498.249,A -85,B 0,C 180,E1 -3933.603,E2 -3933.603} C_VEL
LIN {X 0,Y 537.5,Z 497.144,A -85,B 0,C 180,E1 -3934.439,E2 -3934.439} C_VEL
LIN {X 0,Y 537.538,Z 494.45,A -85,B 0,C 180,E1 -3935.68,E2 -3935.68} C_VEL
LIN {X 0,Y 537.584,Z 490.611,A -85,B 0,C 180,E1 -3936.909,E2 -3936.909} C_VEL
LIN {X 0,Y 537.645,Z 485.571,A -85,B 0,C 180,E1 -3938.123,E2 -3938.123} C_VEL
LIN {X 0,Y 537.719,Z 480.277,A -85,B 0,C 180,E1 -3939.136,E2 -3939.136} C_VEL
LIN {X 0,Y 537.861,Z 473.715,A -85,B 0,C 180,E1 -3940.165,E2 -3940.165} C_VEL
LIN {X 0,Y 538.023,Z 466.2,A -85,B 0,C 180,E1 -3941.138,E2 -3941.138} C_VEL
LIN {X 0,Y 538.275,Z 455.709,A -85,B 0,C 180,E1 -3942.231,E2 -3942.231} C_VEL
LIN {X 0,Y 538.438,Z 446.296,A -85,B 0,C 180,E1 -3943.02,E2 -3943.02} C_VEL
LIN {X 0,Y 538.702,Z 436.155,A -85,B 0,C 180,E1 -3943.711,E2 -3943.711} C_VEL
LIN {X 0,Y 538.877,Z 425.504,A -85,B 0,C 180,E1 -3944.295,E2 -3944.295} C_VEL
LIN {X 0,Y 539.014,Z 415.123,A -85,B 0,C 180,E1 -3944.739,E2 -3944.739} C_VEL
LIN {X 0,Y 539.156,Z 402.608,A -85,B 0,C 180,E1 -3945.13,E2 -3945.13} C_VEL
LIN {X 0,Y 539.308,Z 389.862,A -85,B 0,C 180,E1 -3945.376,E2 -3945.376} C_VEL
LIN {X 0,Y 539.614,Z 297.653,A -85,B 0,C 180,E1 -3946.622,E2 -3946.622} C_VEL
LIN {X 0,Y 538.083,Z 289.182,A -85,B 0,C 180,E1 -3946.787,E2 -3946.787} C_VEL
LIN {X 0,Y 538.021,Z 273.469,A -85,B 0,C 180,E1 -3949.415,E2 -3949.415} C_VEL
LIN {X 0,Y 538.026,Z 273.467,A -85,B 0,C 180,E1 -3952.495,E2 -3952.495} C_VEL
LIN {X 0,Y 538.126,Z 273.458,A -85,B 0,C 180,E1 -3954.755,E2 -3954.755} C_VEL
LIN {X 0,Y 538.102,Z 273.454,A -85,B 0,C 180,E1 -3957.755,E2 -3957.755} C_VEL
LIN {X 0,Y 538.131,Z 273.455,A -85,B 0,C 180,E1 -3960.749,E2 -3960.749} C_VEL
LIN {X 0,Y 538.089,Z 273.462,A -85,B 0,C 180,E1 -3962.995,E2 -3962.995} C_VEL
LIN {X 0,Y 538.066,Z 273.456,A -85,B 0,C 180,E1 -3965.998,E2 -3965.998} C_VEL
LIN {X 0,Y 538.023,Z 273.471,A -85,B 0,C 180,E1 -3969.019,E2 -3969.019} C_VEL
LIN {X 0,Y 538.026,Z 273.461,A -85,B 0,C 180,E1 -3972.064,E2 -3972.064} C_VEL
LIN {X 0,Y 537.999,Z 273.472,A -85,B 0,C 180,E1 -3975.145,E2 -3975.145} C_VEL
LIN {X 0,Y 537.984,Z 273.466,A -85,B 0,C 180,E1 -3978.272,E2 -3978.272} C_VEL
LIN {X 0,Y 537.988,Z 273.468,A -85,B 0,C 180,E1 -3980.654,E2 -3980.654} C_VEL
LIN {X 0,Y 537.971,Z 273.468,A -85,B 0,C 180,E1 -3983.89,E2 -3983.89} C_VEL
LIN {X 0,Y 538.001,Z 273.463,A -85,B 0,C 180,E1 -3986.369,E2 -3986.369} C_VEL
LIN {X 0,Y 537.983,Z 273.473,A -85,B 0,C 180,E1 -3988.937,E2 -3988.937} C_VEL
LIN {X 0,Y 537.981,Z 273.466,A -85,B 0,C 180,E1 -3991.894,E2 -3991.894} C_VEL
LIN {X 0,Y 537.989,Z 273.467,A -85,B 0,C 180,E1 -3994.625,E2 -3994.625} C_VEL
LIN {X 0,Y 537.966,Z 273.476,A -85,B 0,C 180,E1 -3997.174,E2 -3997.174} C_VEL
LIN {X 0,Y 538.016,Z 273.464,A -85,B 0,C 180,E1 -3999.798,E2 -3999.798} C_VEL
LIN {X 0,Y 537.985,Z 273.468,A -85,B 0,C 180,E1 -4002.79,E2 -4002.79} C_VEL
LIN {X 0,Y 537.997,Z 273.466,A -85,B 0,C 180,E1 -4005.929,E2 -4005.929} C_VEL
LIN {X 0,Y 538.024,Z 273.47,A -85,B 0,C 180,E1 -4009.256,E2 -4009.256} C_VEL
LIN {X 0,Y 537.966,Z 273.469,A -85,B 0,C 180,E1 -4012.126,E2 -4012.126} C_VEL
LIN {X 0,Y 537.976,Z 273.472,A -85,B 0,C 180,E1 -4014.92,E2 -4014.92} C_VEL
LIN {X 0,Y 537.999,Z 273.473,A -85,B 0,C 180,E1 -4017.621,E2 -4017.621} C_VEL
LIN {X 0,Y 537.999,Z 273.467,A -85,B 0,C 180,E1 -4020.242,E2 -4020.242} C_VEL
LIN {X 0,Y 538.017,Z 273.466,A -85,B 0,C 180,E1 -4022.798,E2 -4022.798} C_VEL
LIN {X 0,Y 538.085,Z 273.577,A -85,B 0,C 180,E1 -4025.273,E2 -4025.273} C_VEL
LIN {X 0,Y 539.107,Z 279.735,A -85,B 0,C 180,E1 -4026.167,E2 -4026.167} C_VEL
LIN {X 0,Y 538.969,Z 298.685,A -85,B 0,C 180,E1 -4028.79,E2 -4028.79} C_VEL
LIN {X 0,Y 538.653,Z 321.105,A -85,B 0,C 180,E1 -4031.912,E2 -4031.912} C_VEL
LIN {X 0,Y 538.355,Z 342.594,A -85,B 0,C 180,E1 -4034.868,E2 -4034.868} C_VEL
LIN {X 0,Y 538.32,Z 345.38,A -85,B 0,C 180,E1 -4035.247,E2 -4035.247} C_VEL
LIN {X 0,Y 539.637,Z 356.3,A -85,B 0,C 180,E1 -4035.433,E2 -4035.433} C_VEL
LIN {X 0,Y 539.272,Z 454.886,A -85,B 0,C 180,E1 -4036.771,E2 -4036.771} C_VEL
LIN {X 0,Y 539.08,Z 468.02,A -85,B 0,C 180,E1 -4037.102,E2 -4037.102} C_VEL
LIN {X 0,Y 538.884,Z 480.711,A -85,B 0,C 180,E1 -4037.576,E2 -4037.576} C_VEL
LIN {X 0,Y 538.686,Z 492.896,A -85,B 0,C 180,E1 -4038.198,E2 -4038.198} C_VEL
LIN {X 0,Y 538.452,Z 505.006,A -85,B 0,C 180,E1 -4038.998,E2 -4038.998} C_VEL
LIN {X 0,Y 538.199,Z 515.291,A -85,B 0,C 180,E1 -4039.849,E2 -4039.849} C_VEL
LIN {X 0,Y 538.005,Z 524.538,A -85,B 0,C 180,E1 -4040.794,E2 -4040.794} C_VEL
LIN {X 0,Y 537.849,Z 533.546,A -85,B 0,C 180,E1 -4041.927,E2 -4041.927} C_VEL
LIN {X 0,Y 537.706,Z 540.792,A -85,B 0,C 180,E1 -4043.058,E2 -4043.058} C_VEL
LIN {X 0,Y 537.692,Z 545.675,A -85,B 0,C 180,E1 -4044,E2 -4044} C_VEL
LIN {X 0,Y 537.54,Z 550.379,A -85,B 0,C 180,E1 -4045.127,E2 -4045.127} C_VEL
LIN {X 0,Y 537.591,Z 553.962,A -85,B 0,C 180,E1 -4046.254,E2 -4046.254} C_VEL
LIN {X 0,Y 537.551,Z 555.81,A -85,B 0,C 180,E1 -4047.004,E2 -4047.004} C_VEL
LIN {X 0,Y 537.451,Z 558.183,A -85,B 0,C 180,E1 -4048.503,E2 -4048.503} C_VEL
LIN {X 0,Y 537.442,Z 559,A -85,B 0,C 180,E1 -4050.001,E2 -4050.001} C_VEL
LIN {X 0,Y 537.451,Z 558.182,A -85,B 0,C 180,E1 -4051.5,E2 -4051.5} C_VEL
LIN {X 0,Y 537.551,Z 555.808,A -85,B 0,C 180,E1 -4052.999,E2 -4052.999} C_VEL
LIN {X 0,Y 537.604,Z 552.893,A -85,B 0,C 180,E1 -4054.124,E2 -4054.124} C_VEL
LIN {X 0,Y 537.588,Z 548.945,A -85,B 0,C 180,E1 -4055.251,E2 -4055.251} C_VEL
LIN {X 0,Y 537.649,Z 544.053,A -85,B 0,C 180,E1 -4056.335,E2 -4056.335} C_VEL
LIN {X 0,Y 537.773,Z 537.36,A -85,B 0,C 180,E1 -4057.51,E2 -4057.51} C_VEL
LIN {X 0,Y 537.937,Z 529.284,A -85,B 0,C 180,E1 -4058.641,E2 -4058.641} C_VEL
LIN {X 0,Y 538.116,Z 521.054,A -85,B 0,C 180,E1 -4059.586,E2 -4059.586} C_VEL
LIN {X 0,Y 538.342,Z 511.016,A -85,B 0,C 180,E1 -4060.531,E2 -4060.531} C_VEL
LIN {X 0,Y 538.54,Z 501.103,A -85,B 0,C 180,E1 -4061.289,E2 -4061.289} C_VEL
LIN {X 0,Y 538.733,Z 489.898,A -85,B 0,C 180,E1 -4061.975,E2 -4061.975} C_VEL
LIN {X 0,Y 538.926,Z 477.356,A -85,B 0,C 180,E1 -4062.569,E2 -4062.569} C_VEL
LIN {X 0,Y 539.128,Z 465.005,A -85,B 0,C 180,E1 -4062.995,E2 -4062.995} C_VEL
LIN {X 0,Y 539.295,Z 452.303,A -85,B 0,C 180,E1 -4063.278,E2 -4063.278} C_VEL
LIN {X 0,Y 539.525,Z 353.569,A -85,B 0,C 180,E1 -4064.608,E2 -4064.608} C_VEL
LIN {X 0,Y 538.398,Z 345.713,A -85,B 0,C 180,E1 -4064.758,E2 -4064.758} C_VEL
LIN {X 0,Y 538.719,Z 323.049,A -85,B 0,C 180,E1 -4067.94,E2 -4067.94} C_VEL
LIN {X 0,Y 539.153,Z 300.038,A -85,B 0,C 180,E1 -4071.205,E2 -4071.205} C_VEL
LIN {X 0,Y 539.499,Z 282.022,A -85,B 0,C 180,E1 -4073.817,E2 -4073.817} C_VEL
LIN {X 0,Y 538.663,Z 276.47,A -85,B 0,C 180,E1 -4074.676,E2 -4074.676} C_VEL
LIN {X 0,Y 538.042,Z 273.466,A -85,B 0,C 180,E1 -4075.171,E2 -4075.171} C_VEL
LIN {X 0,Y 538.005,Z 273.467,A -85,B 0,C 180,E1 -4078.05,E2 -4078.05} C_VEL
LIN {X 0,Y 538,Z 273.473,A -85,B 0,C 180,E1 -4080.626,E2 -4080.626} C_VEL
LIN {X 0,Y 538.012,Z 273.464,A -85,B 0,C 180,E1 -4083.277,E2 -4083.277} C_VEL
LIN {X 0,Y 537.977,Z 273.468,A -85,B 0,C 180,E1 -4086.003,E2 -4086.003} C_VEL
LIN {X 0,Y 537.994,Z 273.471,A -85,B 0,C 180,E1 -4088.829,E2 -4088.829} C_VEL
LIN {X 0,Y 537.981,Z 273.467,A -85,B 0,C 180,E1 -4091.872,E2 -4091.872} C_VEL
LIN {X 0,Y 537.976,Z 273.474,A -85,B 0,C 180,E1 -4094.861,E2 -4094.861} C_VEL
LIN {X 0,Y 537.968,Z 273.47,A -85,B 0,C 180,E1 -4097.209,E2 -4097.209} C_VEL
LIN {X 0,Y 538.006,Z 273.469,A -85,B 0,C 180,E1 -4100.413,E2 -4100.413} C_VEL
LIN {X 0,Y 537.992,Z 273.469,A -85,B 0,C 180,E1 -4103.064,E2 -4103.064} C_VEL
LIN {X 0,Y 537.98,Z 273.467,A -85,B 0,C 180,E1 -4105.824,E2 -4105.824} C_VEL
LIN {X 0,Y 537.979,Z 273.473,A -85,B 0,C 180,E1 -4108.496,E2 -4108.496} C_VEL
LIN {X 0,Y 537.988,Z 273.47,A -85,B 0,C 180,E1 -4111.095,E2 -4111.095} C_VEL
LIN {X 0,Y 537.991,Z 273.466,A -85,B 0,C 180,E1 -4113.63,E2 -4113.63} C_VEL
LIN {X 0,Y 537.971,Z 273.475,A -85,B 0,C 180,E1 -4116.926,E2 -4116.926} C_VEL
LIN {X 0,Y 538.044,Z 273.461,A -85,B 0,C 180,E1 -4120.146,E2 -4120.146} C_VEL
LIN {X 0,Y 537.973,Z 273.47,A -85,B 0,C 180,E1 -4123.297,E2 -4123.297} C_VEL
LIN {X 0,Y 538.017,Z 273.463,A -85,B 0,C 180,E1 -4125.629,E2 -4125.629} C_VEL
LIN {X 0,Y 538.061,Z 273.464,A -85,B 0,C 180,E1 -4128.701,E2 -4128.701} C_VEL
LIN {X 0,Y 538.045,Z 273.459,A -85,B 0,C 180,E1 -4131.739,E2 -4131.739} C_VEL
LIN {X 0,Y 538.124,Z 273.457,A -85,B 0,C 180,E1 -4134.754,E2 -4134.754} C_VEL
LIN {X 0,Y 538.12,Z 273.45,A -85,B 0,C 180,E1 -4137.754,E2 -4137.754} C_VEL
LIN {X 0,Y 538.15,Z 273.453,A -85,B 0,C 180,E1 -4140.748,E2 -4140.748} C_VEL
LIN {X 0,Y 538.105,Z 273.459,A -85,B 0,C 180,E1 -4142.994,E2 -4142.994} C_VEL
LIN {X 0,Y 538.08,Z 273.455,A -85,B 0,C 180,E1 -4145.997,E2 -4145.997} C_VEL
LIN {X 0,Y 538.04,Z 273.467,A -85,B 0,C 180,E1 -4149.018,E2 -4149.018} C_VEL
LIN {X 0,Y 538.046,Z 273.46,A -85,B 0,C 180,E1 -4152.063,E2 -4152.063} C_VEL
LIN {X 0,Y 538.007,Z 273.469,A -85,B 0,C 180,E1 -4155.144,E2 -4155.144} C_VEL
LIN {X 0,Y 538,Z 273.467,A -85,B 0,C 180,E1 -4158.271,E2 -4158.271} C_VEL
LIN {X 0,Y 538.007,Z 273.471,A -85,B 0,C 180,E1 -4160.652,E2 -4160.652} C_VEL
LIN {X 0,Y 537.989,Z 273.466,A -85,B 0,C 180,E1 -4163.889,E2 -4163.889} C_VEL
LIN {X 0,Y 538.017,Z 273.465,A -85,B 0,C 180,E1 -4166.368,E2 -4166.368} C_VEL
LIN {X 0,Y 538.024,Z 273.469,A -85,B 0,C 180,E1 -4168.94,E2 -4168.94} C_VEL
LIN {X 0,Y 537.996,Z 273.466,A -85,B 0,C 180,E1 -4171.892,E2 -4171.892} C_VEL
LIN {X 0,Y 538.006,Z 273.47,A -85,B 0,C 180,E1 -4174.623,E2 -4174.623} C_VEL
LIN {X 0,Y 537.983,Z 273.473,A -85,B 0,C 180,E1 -4177.173,E2 -4177.173} C_VEL
LIN {X 0,Y 538.024,Z 273.463,A -85,B 0,C 180,E1 -4180.291,E2 -4180.291} C_VEL
LIN {X 0,Y 537.373,Z 273.55,A -85,B 0,C 180,E1 -4180.916,E2 -4180.916} C_VEL
LIN {X 0,Y 534.511,Z 273.908,A -85,B 0,C 180,E1 -4181.93,E2 -4181.93} C_VEL
LIN {X 0,Y 532.077,Z 274.21,A -85,B 0,C 180,E1 -4182.747,E2 -4182.747} C_VEL
LIN {X 0,Y 531.026,Z 274.338,A -85,B 0,C 180,E1 -4183.378,E2 -4183.378} C_VEL
LIN {X 0,Y 530.939,Z 274.346,A -85,B 0,C 180,E1 -4183.592,E2 -4183.592} C_VEL
LIN {X 0,Y 530.947,Z 274.347,A -85,B 0,C 180,E1 -4186.507,E2 -4186.507} C_VEL
LIN {X 0,Y 530.991,Z 274.34,A -85,B 0,C 180,E1 -4189.571,E2 -4189.571} C_VEL
LIN {X 0,Y 530.962,Z 274.346,A -85,B 0,C 180,E1 -4192.577,E2 -4192.577} C_VEL
LIN {X 0,Y 530.987,Z 274.343,A -85,B 0,C 180,E1 -4195.313,E2 -4195.313} C_VEL
LIN {X 0,Y 530.955,Z 274.343,A -85,B 0,C 180,E1 -4198.033,E2 -4198.033} C_VEL
LIN {X 0,Y 530.98,Z 274.347,A -85,B 0,C 180,E1 -4200.875,E2 -4200.875} C_VEL
LIN {X 0,Y 530.997,Z 274.343,A -85,B 0,C 180,E1 -4203.258,E2 -4203.258} C_VEL
LIN {X 0,Y 530.978,Z 274.34,A -85,B 0,C 180,E1 -4205.962,E2 -4205.962} C_VEL
LIN {X 0,Y 530.995,Z 274.345,A -85,B 0,C 180,E1 -4209.063,E2 -4209.063} C_VEL
LIN {X 0,Y 531.013,Z 274.336,A -85,B 0,C 180,E1 -4212.278,E2 -4212.278} C_VEL
LIN {X 0,Y 531.016,Z 274.339,A -85,B 0,C 180,E1 -4215.436,E2 -4215.436} C_VEL
LIN {X 0,Y 531.034,Z 274.335,A -85,B 0,C 180,E1 -4218.55,E2 -4218.55} C_VEL
LIN {X 0,Y 531.054,Z 274.332,A -85,B 0,C 180,E1 -4221.629,E2 -4221.629} C_VEL
LIN {X 0,Y 531.118,Z 274.326,A -85,B 0,C 180,E1 -4224.685,E2 -4224.685} C_VEL
LIN {X 0,Y 531.139,Z 274.321,A -85,B 0,C 180,E1 -4227.724,E2 -4227.724} C_VEL
LIN {X 0,Y 531.15,Z 274.323,A -85,B 0,C 180,E1 -4230.757,E2 -4230.757} C_VEL
LIN {X 0,Y 531.103,Z 274.333,A -85,B 0,C 180,E1 -4233.033,E2 -4233.033} C_VEL
LIN {X 0,Y 531.072,Z 274.328,A -85,B 0,C 180,E1 -4236.075,E2 -4236.075} C_VEL
LIN {X 0,Y 531.051,Z 274.331,A -85,B 0,C 180,E1 -4238.369,E2 -4238.369} C_VEL
LIN {X 0,Y 531.06,Z 274.331,A -85,B 0,C 180,E1 -4241.678,E2 -4241.678} C_VEL
LIN {X 0,Y 531.022,Z 274.34,A -85,B 0,C 180,E1 -4244.953,E2 -4244.953} C_VEL
LIN {X 0,Y 531.006,Z 274.337,A -85,B 0,C 180,E1 -4247.72,E2 -4247.72} C_VEL
LIN {X 0,Y 530.993,Z 274.343,A -85,B 0,C 180,E1 -4250.935,E2 -4250.935} C_VEL
LIN {X 0,Y 530.992,Z 274.337,A -85,B 0,C 180,E1 -4254.042,E2 -4254.042} C_VEL
LIN {X 0,Y 530.996,Z 274.34,A -85,B 0,C 180,E1 -4256.74,E2 -4256.74} C_VEL
LIN {X 0,Y 530.98,Z 274.346,A -85,B 0,C 180,E1 -4259.318,E2 -4259.318} C_VEL
LIN {X 0,Y 530.959,Z 274.341,A -85,B 0,C 180,E1 -4262.1,E2 -4262.1} C_VEL
LIN {X 0,Y 530.967,Z 274.344,A -85,B 0,C 180,E1 -4264.851,E2 -4264.851} C_VEL
LIN {X 0,Y 530.946,Z 274.348,A -85,B 0,C 180,E1 -4267.503,E2 -4267.503} C_VEL
LIN {X 0,Y 530.997,Z 274.338,A -85,B 0,C 180,E1 -4270.425,E2 -4270.425} C_VEL
LIN {X 0,Y 531.064,Z 274.335,A -85,B 0,C 180,E1 -4274.003,E2 -4274.003} C_VEL
LIN {X 0,Y 531.267,Z 279.107,A -85,B 0,C 180,E1 -4274.993,E2 -4274.993} C_VEL
LIN {X 0,Y 531.162,Z 289.762,A -85,B 0,C 180,E1 -4277.104,E2 -4277.104} C_VEL
LIN {X 0,Y 532.797,Z 299.112,A -85,B 0,C 180,E1 -4277.298,E2 -4277.298} C_VEL
LIN {X 0,Y 532.37,Z 396.374,A -85,B 0,C 180,E1 -4278.648,E2 -4278.648} C_VEL
LIN {X 0,Y 532.238,Z 409.9,A -85,B 0,C 180,E1 -4278.997,E2 -4278.997} C_VEL
LIN {X 0,Y 532,Z 422.381,A -85,B 0,C 180,E1 -4279.475,E2 -4279.475} C_VEL
LIN {X 0,Y 531.758,Z 434.275,A -85,B 0,C 180,E1 -4280.098,E2 -4280.098} C_VEL
LIN {X 0,Y 531.532,Z 443.62,A -85,B 0,C 180,E1 -4280.711,E2 -4280.711} C_VEL
LIN {X 0,Y 531.344,Z 452.961,A -85,B 0,C 180,E1 -4281.458,E2 -4281.458} C_VEL
LIN {X 0,Y 531.11,Z 462.498,A -85,B 0,C 180,E1 -4282.385,E2 -4282.385} C_VEL
LIN {X 0,Y 530.926,Z 471.319,A -85,B 0,C 180,E1 -4283.44,E2 -4283.44} C_VEL
LIN {X 0,Y 530.717,Z 479.04,A -85,B 0,C 180,E1 -4284.586,E2 -4284.586} C_VEL
LIN {X 0,Y 530.598,Z 485.254,A -85,B 0,C 180,E1 -4285.742,E2 -4285.742} C_VEL
LIN {X 0,Y 530.54,Z 489.916,A -85,B 0,C 180,E1 -4286.828,E2 -4286.828} C_VEL
LIN {X 0,Y 530.475,Z 493.813,A -85,B 0,C 180,E1 -4287.999,E2 -4287.999} C_VEL
LIN {X 0,Y 530.45,Z 496.101,A -85,B 0,C 180,E1 -4288.888,E2 -4288.888} C_VEL
LIN {X 0,Y 530.408,Z 497.779,A -85,B 0,C 180,E1 -4289.768,E2 -4289.768} C_VEL
LIN {X 0,Y 530.382,Z 499.163,A -85,B 0,C 180,E1 -4290.979,E2 -4290.979} C_VEL
LIN {X 0,Y 530.344,Z 499.405,A -85,B 0,C 180,E1 -4292.593,E2 -4292.593} C_VEL
LIN {X 0,Y 530.358,Z 499.097,A -85,B 0,C 180,E1 -4293.222,E2 -4293.222} C_VEL
LIN {X 0,Y 530.409,Z 497.861,A -85,B 0,C 180,E1 -4294.276,E2 -4294.276} C_VEL
LIN {X 0,Y 530.46,Z 494.795,A -85,B 0,C 180,E1 -4295.751,E2 -4295.751} C_VEL
LIN {X 0,Y 530.533,Z 490.929,A -85,B 0,C 180,E1 -4296.997,E2 -4296.997} C_VEL
LIN {X 0,Y 530.587,Z 485.848,A -85,B 0,C 180,E1 -4298.231,E2 -4298.231} C_VEL
LIN {X 0,Y 530.752,Z 479.366,A -85,B 0,C 180,E1 -4299.458,E2 -4299.458} C_VEL
LIN {X 0,Y 530.914,Z 471.209,A -85,B 0,C 180,E1 -4300.675,E2 -4300.675} C_VEL
LIN {X 0,Y 531.115,Z 462.783,A -85,B 0,C 180,E1 -4301.684,E2 -4301.684} C_VEL
LIN {X 0,Y 531.327,Z 453.58,A -85,B 0,C 180,E1 -4302.587,E2 -4302.587} C_VEL
LIN {X 0,Y 531.595,Z 443.586,A -85,B 0,C 180,E1 -4303.388,E2 -4303.388} C_VEL
LIN {X 0,Y 531.839,Z 432.815,A -85,B 0,C 180,E1 -4304.086,E2 -4304.086} C_VEL
LIN {X 0,Y 532.074,Z 419.91,A -85,B 0,C 180,E1 -4304.724,E2 -4304.724} C_VEL
LIN {X 0,Y 532.205,Z 407.28,A -85,B 0,C 180,E1 -4305.176,E2 -4305.176} C_VEL
LIN {X 0,Y 532.342,Z 394.624,A -85,B 0,C 180,E1 -4305.473,E2 -4305.473} C_VEL
LIN {X 0,Y 532.725,Z 298.302,A -85,B 0,C 180,E1 -4306.81,E2 -4306.81} C_VEL
LIN {X 0,Y 531.077,Z 289.21,A -85,B 0,C 180,E1 -4306.999,E2 -4306.999} C_VEL
LIN {X 0,Y 530.988,Z 274.345,A -85,B 0,C 180,E1 -4309.466,E2 -4309.466} C_VEL
LIN {X 0,Y 531.003,Z 274.341,A -85,B 0,C 180,E1 -4312.395,E2 -4312.395} C_VEL
LIN {X 0,Y 531.081,Z 274.335,A -85,B 0,C 180,E1 -4314.685,E2 -4314.685} C_VEL
LIN {X 0,Y 531.075,Z 274.329,A -85,B 0,C 180,E1 -4317.725,E2 -4317.725} C_VEL
LIN {X 0,Y 531.1,Z 274.331,A -85,B 0,C 180,E1 -4320.759,E2 -4320.759} C_VEL
LIN {X 0,Y 531.054,Z 274.338,A -85,B 0,C 180,E1 -4323.035,E2 -4323.035} C_VEL
LIN {X 0,Y 531.025,Z 274.334,A -85,B 0,C 180,E1 -4326.078,E2 -4326.078} C_VEL
LIN {X 0,Y 530.983,Z 274.346,A -85,B 0,C 180,E1 -4329.139,E2 -4329.139} C_VEL
LIN {X 0,Y 531.007,Z 274.337,A -85,B 0,C 180,E1 -4331.682,E2 -4331.682} C_VEL
LIN {X 0,Y 530.99,Z 274.345,A -85,B 0,C 180,E1 -4334.965,E2 -4334.965} C_VEL
LIN {X 0,Y 530.96,Z 274.341,A -85,B 0,C 180,E1 -4337.725,E2 -4337.725} C_VEL
LIN {X 0,Y 530.97,Z 274.339,A -85,B 0,C 180,E1 -4340.13,E2 -4340.13} C_VEL
LIN {X 0,Y 530.912,Z 274.352,A -85,B 0,C 180,E1 -4343.399,E2 -4343.399} C_VEL
LIN {X 0,Y 530.966,Z 274.34,A -85,B 0,C 180,E1 -4345.9,E2 -4345.9} C_VEL
LIN {X 0,Y 530.951,Z 274.343,A -85,B 0,C 180,E1 -4348.459,E2 -4348.459} C_VEL
LIN {X 0,Y 530.917,Z 274.355,A -85,B 0,C 180,E1 -4351.082,E2 -4351.082} C_VEL
LIN {X 0,Y 530.948,Z 274.343,A -85,B 0,C 180,E1 -4353.776,E2 -4353.776} C_VEL
LIN {X 0,Y 530.925,Z 274.347,A -85,B 0,C 180,E1 -4356.561,E2 -4356.561} C_VEL
LIN {X 0,Y 530.968,Z 274.341,A -85,B 0,C 180,E1 -4359.861,E2 -4359.861} C_VEL
LIN {X 0,Y 530.95,Z 274.342,A -85,B 0,C 180,E1 -4362.46,E2 -4362.46} C_VEL
LIN {X 0,Y 530.956,Z 274.346,A -85,B 0,C 180,E1 -4365.625,E2 -4365.625} C_VEL
LIN {X 0,Y 530.971,Z 274.341,A -85,B 0,C 180,E1 -4368.569,E2 -4368.569} C_VEL
LIN {X 0,Y 530.93,Z 274.351,A -85,B 0,C 180,E1 -4371.533,E2 -4371.533} C_VEL
LIN {X 0,Y 530.931,Z 274.346,A -85,B 0,C 180,E1 -4374.384,E2 -4374.384} C_VEL
LIN {X 0,Y 530.947,Z 274.352,A -85,B 0,C 180,E1 -4377.137,E2 -4377.137} C_VEL
LIN {X 0,Y 530.952,Z 274.348,A -85,B 0,C 180,E1 -4379.807,E2 -4379.807} C_VEL
LIN {X 0,Y 530.961,Z 274.344,A -85,B 0,C 180,E1 -4382.479,E2 -4382.479} C_VEL
LIN {X 0,Y 531.061,Z 274.511,A -85,B 0,C 180,E1 -4385.159,E2 -4385.159} C_VEL
LIN {X 0,Y 532.16,Z 281.988,A -85,B 0,C 180,E1 -4386.251,E2 -4386.251} C_VEL
LIN {X 0,Y 531.973,Z 302.407,A -85,B 0,C 180,E1 -4389.106,E2 -4389.106} C_VEL
LIN {X 0,Y 531.563,Z 325.089,A -85,B 0,C 180,E1 -4392.3,E2 -4392.3} C_VEL
LIN {X 0,Y 531.32,Z 344.867,A -85,B 0,C 180,E1 -4395.041,E2 -4395.041} C_VEL
LIN {X 0,Y 532.745,Z 356.439,A -85,B 0,C 180,E1 -4395.252,E2 -4395.252} C_VEL
LIN {X 0,Y 532.352,Z 453.966,A -85,B 0,C 180,E1 -4396.596,E2 -4396.596} C_VEL
LIN {X 0,Y 532.153,Z 467.253,A -85,B 0,C 180,E1 -4396.931,E2 -4396.931} C_VEL
LIN {X 0,Y 531.911,Z 480.026,A -85,B 0,C 180,E1 -4397.41,E2 -4397.41} C_VEL
LIN {X 0,Y 531.704,Z 492.174,A -85,B 0,C 180,E1 -4398.034,E2 -4398.034} C_VEL
LIN {X 0,Y 531.44,Z 504.436,A -85,B 0,C 180,E1 -4398.851,E2 -4398.851} C_VEL
LIN {X 0,Y 531.177,Z 514.761,A -85,B 0,C 180,E1 -4399.713,E2 -4399.713} C_VEL
LIN {X 0,Y 530.959,Z 524.034,A -85,B 0,C 180,E1 -4400.671,E2 -4400.671} C_VEL
LIN {X 0,Y 530.784,Z 533.063,A -85,B 0,C 180,E1 -4401.819,E2 -4401.819} C_VEL
LIN {X 0,Y 530.631,Z 540.333,A -85,B 0,C 180,E1 -4402.965,E2 -4402.965} C_VEL
LIN {X 0,Y 530.59,Z 546.952,A -85,B 0,C 180,E1 -4404.301,E2 -4404.301} C_VEL
LIN {X 0,Y 530.455,Z 551.321,A -85,B 0,C 180,E1 -4405.442,E2 -4405.442} C_VEL
LIN {X 0,Y 530.516,Z 553.64,A -85,B 0,C 180,E1 -4406.204,E2 -4406.204} C_VEL
LIN {X 0,Y 530.457,Z 555.516,A -85,B 0,C 180,E1 -4406.964,E2 -4406.964} C_VEL
LIN {X 0,Y 530.411,Z 556.92,A -85,B 0,C 180,E1 -4407.723,E2 -4407.723} C_VEL
LIN {X 0,Y 530.346,Z 558.533,A -85,B 0,C 180,E1 -4409.242,E2 -4409.242} C_VEL
LIN {X 0,Y 530.347,Z 558.752,A -85,B 0,C 180,E1 -4410.001,E2 -4410.001} C_VEL
LIN {X 0,Y 530.361,Z 557.925,A -85,B 0,C 180,E1 -4411.52,E2 -4411.52} C_VEL
LIN {X 0,Y 530.411,Z 556.926,A -85,B 0,C 180,E1 -4412.279,E2 -4412.279} C_VEL
LIN {X 0,Y 530.457,Z 555.524,A -85,B 0,C 180,E1 -4413.039,E2 -4413.039} C_VEL
LIN {X 0,Y 530.523,Z 552.572,A -85,B 0,C 180,E1 -4414.179,E2 -4414.179} C_VEL
LIN {X 0,Y 530.525,Z 548.569,A -85,B 0,C 180,E1 -4415.321,E2 -4415.321} C_VEL
LIN {X 0,Y 530.599,Z 542.81,A -85,B 0,C 180,E1 -4416.582,E2 -4416.582} C_VEL
LIN {X 0,Y 530.72,Z 535.687,A -85,B 0,C 180,E1 -4417.802,E2 -4417.802} C_VEL
LIN {X 0,Y 530.913,Z 527.342,A -85,B 0,C 180,E1 -4418.949,E2 -4418.949} C_VEL
LIN {X 0,Y 531.094,Z 518.776,A -85,B 0,C 180,E1 -4419.906,E2 -4419.906} C_VEL
LIN {X 0,Y 531.348,Z 508.196,A -85,B 0,C 180,E1 -4420.864,E2 -4420.864} C_VEL
LIN {X 0,Y 531.6,Z 497.138,A -85,B 0,C 180,E1 -4421.671,E2 -4421.671} C_VEL
LIN {X 0,Y 531.859,Z 486.232,A -85,B 0,C 180,E1 -4422.303,E2 -4422.303} C_VEL
LIN {X 0,Y 532.022,Z 474.352,A -85,B 0,C 180,E1 -4422.832,E2 -4422.832} C_VEL
LIN {X 0,Y 532.233,Z 460.657,A -85,B 0,C 180,E1 -4423.264,E2 -4423.264} C_VEL
LIN {X 0,Y 532.377,Z 448.415,A -85,B 0,C 180,E1 -4423.503,E2 -4423.503} C_VEL
LIN {X 0,Y 532.613,Z 354.197,A -85,B 0,C 180,E1 -4424.787,E2 -4424.787} C_VEL
LIN {X 0,Y 531.356,Z 345.347,A -85,B 0,C 180,E1 -4424.959,E2 -4424.959} C_VEL
LIN {X 0,Y 531.708,Z 324.838,A -85,B 0,C 180,E1 -4427.883,E2 -4427.883} C_VEL
LIN {X 0,Y 532.198,Z 301.116,A -85,B 0,C 180,E1 -4431.293,E2 -4431.293} C_VEL
LIN {X 0,Y 532.58,Z 283.137,A -85,B 0,C 180,E1 -4433.939,E2 -4433.939} C_VEL
LIN {X 0,Y 530.997,Z 274.343,A -85,B 0,C 180,E1 -4435.371,E2 -4435.371} C_VEL
LIN {X 0,Y 530.959,Z 274.35,A -85,B 0,C 180,E1 -4438.456,E2 -4438.456} C_VEL
LIN {X 0,Y 530.945,Z 274.346,A -85,B 0,C 180,E1 -4441.078,E2 -4441.078} C_VEL
LIN {X 0,Y 530.941,Z 274.343,A -85,B 0,C 180,E1 -4443.774,E2 -4443.774} C_VEL
LIN {X 0,Y 530.924,Z 274.354,A -85,B 0,C 180,E1 -4446.558,E2 -4446.558} C_VEL
LIN {X 0,Y 530.954,Z 274.342,A -85,B 0,C 180,E1 -4449.443,E2 -4449.443} C_VEL
LIN {X 0,Y 530.914,Z 274.353,A -85,B 0,C 180,E1 -4452.459,E2 -4452.459} C_VEL
LIN {X 0,Y 530.949,Z 274.343,A -85,B 0,C 180,E1 -4455.449,E2 -4455.449} C_VEL
LIN {X 0,Y 530.941,Z 274.351,A -85,B 0,C 180,E1 -4458.559,E2 -4458.559} C_VEL
LIN {X 0,Y 530.927,Z 274.346,A -85,B 0,C 180,E1 -4461.526,E2 -4461.526} C_VEL
LIN {X 0,Y 530.923,Z 274.351,A -85,B 0,C 180,E1 -4464.377,E2 -4464.377} C_VEL
LIN {X 0,Y 530.938,Z 274.347,A -85,B 0,C 180,E1 -4467.131,E2 -4467.131} C_VEL
LIN {X 0,Y 530.923,Z 274.346,A -85,B 0,C 180,E1 -4469.8,E2 -4469.8} C_VEL
LIN {X 0,Y 530.976,Z 274.345,A -85,B 0,C 180,E1 -4472.467,E2 -4472.467} C_VEL
LIN {X 0,Y 530.915,Z 274.353,A -85,B 0,C 180,E1 -4474.938,E2 -4474.938} C_VEL
LIN {X 0,Y 530.941,Z 274.344,A -85,B 0,C 180,E1 -4477.897,E2 -4477.897} C_VEL
LIN {X 0,Y 530.947,Z 274.35,A -85,B 0,C 180,E1 -4480.675,E2 -4480.675} C_VEL
LIN {X 0,Y 530.932,Z 274.35,A -85,B 0,C 180,E1 -4483.069,E2 -4483.069} C_VEL
LIN {X 0,Y 530.975,Z 274.341,A -85,B 0,C 180,E1 -4485.434,E2 -4485.434} C_VEL
LIN {X 0,Y 531.014,Z 274.341,A -85,B 0,C 180,E1 -4488.549,E2 -4488.549} C_VEL
LIN {X 0,Y 531.015,Z 274.335,A -85,B 0,C 180,E1 -4491.628,E2 -4491.628} C_VEL
LIN {X 0,Y 531.082,Z 274.333,A -85,B 0,C 180,E1 -4494.685,E2 -4494.685} C_VEL
LIN {X 0,Y 531.093,Z 274.326,A -85,B 0,C 180,E1 -4497.724,E2 -4497.724} C_VEL
LIN {X 0,Y 531.12,Z 274.329,A -85,B 0,C 180,E1 -4500.758,E2 -4500.758} C_VEL
LIN {X 0,Y 531.071,Z 274.334,A -85,B 0,C 180,E1 -4503.034,E2 -4503.034} C_VEL
LIN {X 0,Y 531.036,Z 274.333,A -85,B 0,C 180,E1 -4506.077,E2 -4506.077} C_VEL
LIN {X 0,Y 531,Z 274.342,A -85,B 0,C 180,E1 -4509.138,E2 -4509.138} C_VEL
LIN {X 0,Y 531.027,Z 274.334,A -85,B 0,C 180,E1 -4511.681,E2 -4511.681} C_VEL
LIN {X 0,Y 530.991,Z 274.346,A -85,B 0,C 180,E1 -4514.956,E2 -4514.956} C_VEL
LIN {X 0,Y 530.979,Z 274.34,A -85,B 0,C 180,E1 -4517.723,E2 -4517.723} C_VEL
LIN {X 0,Y 530.966,Z 274.348,A -85,B 0,C 180,E1 -4520.939,E2 -4520.939} C_VEL
LIN {X 0,Y 530.945,Z 274.345,A -85,B 0,C 180,E1 -4524.226,E2 -4524.226} C_VEL
LIN {X 0,Y 530.978,Z 274.347,A -85,B 0,C 180,E1 -4526.745,E2 -4526.745} C_VEL
LIN {X 0,Y 530.969,Z 274.345,A -85,B 0,C 180,E1 -4529.323,E2 -4529.323} C_VEL
LIN {X 0,Y 530.949,Z 274.344,A -85,B 0,C 180,E1 -4532.104,E2 -4532.104} C_VEL
LIN {X 0,Y 530.963,Z 274.349,A -85,B 0,C 180,E1 -4534.856,E2 -4534.856} C_VEL
LIN {X 0,Y 530.941,Z 274.346,A -85,B 0,C 180,E1 -4537.509,E2 -4537.509} C_VEL
LIN {X 0,Y 530.984,Z 274.342,A -85,B 0,C 180,E1 -4540.432,E2 -4540.432} C_VEL
LIN {X 0,Y 530.942,Z 274.347,A -85,B 0,C 180,E1 -4543.496,E2 -4543.496} C_VEL
LIN {X 0,Y 530.939,Z 274.346,A -85,B 0,C 180,E1 -4543.592,E2 -4543.592} C_VEL
LIN {X 0,Y 530.268,Z 274.43,A -85,B 0,C 180,E1 -4544.226,E2 -4544.226} C_VEL
LIN {X 0,Y 527.422,Z 274.789,A -85,B 0,C 180,E1 -4545.255,E2 -4545.255} C_VEL
LIN {X 0,Y 525.019,Z 275.092,A -85,B 0,C 180,E1 -4546.083,E2 -4546.083} C_VEL
LIN {X 0,Y 523.988,Z 275.218,A -85,B 0,C 180,E1 -4546.723,E2 -4546.723} C_VEL
LIN {X 0,Y 523.903,Z 275.227,A -85,B 0,C 180,E1 -4546.94,E2 -4546.94} C_VEL
LIN {X 0,Y 523.962,Z 275.214,A -85,B 0,C 180,E1 -4549.925,E2 -4549.925} C_VEL
LIN {X 0,Y 523.903,Z 275.228,A -85,B 0,C 180,E1 -4552.87,E2 -4552.87} C_VEL
LIN {X 0,Y 523.93,Z 275.219,A -85,B 0,C 180,E1 -4555.712,E2 -4555.712} C_VEL
LIN {X 0,Y 523.909,Z 275.223,A -85,B 0,C 180,E1 -4558.457,E2 -4558.457} C_VEL
LIN {X 0,Y 523.931,Z 275.224,A -85,B 0,C 180,E1 -4561.127,E2 -4561.127} C_VEL
LIN {X 0,Y 523.976,Z 275.212,A -85,B 0,C 180,E1 -4563.981,E2 -4563.981} C_VEL
LIN {X 0,Y 523.919,Z 275.22,A -85,B 0,C 180,E1 -4566.271,E2 -4566.271} C_VEL
LIN {X 0,Y 523.94,Z 275.222,A -85,B 0,C 180,E1 -4568.767,E2 -4568.767} C_VEL
LIN {X 0,Y 523.947,Z 275.221,A -85,B 0,C 180,E1 -4571.221,E2 -4571.221} C_VEL
LIN {X 0,Y 523.933,Z 275.219,A -85,B 0,C 180,E1 -4573.639,E2 -4573.639} C_VEL
LIN {X 0,Y 523.936,Z 275.217,A -85,B 0,C 180,E1 -4576.028,E2 -4576.028} C_VEL
LIN {X 0,Y 524.01,Z 275.209,A -85,B 0,C 180,E1 -4578.394,E2 -4578.394} C_VEL
LIN {X 0,Y 524.002,Z 275.212,A -85,B 0,C 180,E1 -4581.516,E2 -4581.516} C_VEL
LIN {X 0,Y 524.079,Z 275.202,A -85,B 0,C 180,E1 -4584.613,E2 -4584.613} C_VEL
LIN {X 0,Y 524.111,Z 275.197,A -85,B 0,C 180,E1 -4587.693,E2 -4587.693} C_VEL
LIN {X 0,Y 524.12,Z 275.198,A -85,B 0,C 180,E1 -4590.767,E2 -4590.767} C_VEL
LIN {X 0,Y 524.07,Z 275.208,A -85,B 0,C 180,E1 -4593.073,E2 -4593.073} C_VEL
LIN {X 0,Y 524.033,Z 275.205,A -85,B 0,C 180,E1 -4596.157,E2 -4596.157} C_VEL
LIN {X 0,Y 523.999,Z 275.21,A -85,B 0,C 180,E1 -4598.482,E2 -4598.482} C_VEL
LIN {X 0,Y 524.018,Z 275.208,A -85,B 0,C 180,E1 -4601.749,E2 -4601.749} C_VEL
LIN {X 0,Y 523.984,Z 275.219,A -85,B 0,C 180,E1 -4605.05,E2 -4605.05} C_VEL
LIN {X 0,Y 523.954,Z 275.215,A -85,B 0,C 180,E1 -4607.966,E2 -4607.966} C_VEL
LIN {X 0,Y 523.961,Z 275.214,A -85,B 0,C 180,E1 -4610.407,E2 -4610.407} C_VEL
LIN {X 0,Y 523.93,Z 275.222,A -85,B 0,C 180,E1 -4612.889,E2 -4612.889} C_VEL
LIN {X 0,Y 523.969,Z 275.212,A -85,B 0,C 180,E1 -4616.017,E2 -4616.017} C_VEL
LIN {X 0,Y 523.932,Z 275.221,A -85,B 0,C 180,E1 -4618.871,E2 -4618.871} C_VEL
LIN {X 0,Y 523.911,Z 275.223,A -85,B 0,C 180,E1 -4621.54,E2 -4621.54} C_VEL
LIN {X 0,Y 523.922,Z 275.218,A -85,B 0,C 180,E1 -4624.286,E2 -4624.286} C_VEL
LIN {X 0,Y 523.89,Z 275.23,A -85,B 0,C 180,E1 -4627.128,E2 -4627.128} C_VEL
LIN {X 0,Y 523.963,Z 275.214,A -85,B 0,C 180,E1 -4630.134,E2 -4630.134} C_VEL
LIN {X 0,Y 524,Z 275.217,A -85,B 0,C 180,E1 -4633.593,E2 -4633.593} C_VEL
LIN {X 0,Y 524.02,Z 275.222,A -85,B 0,C 180,E1 -4633.928,E2 -4633.928} C_VEL
LIN {X 0,Y 524.326,Z 279.162,A -85,B 0,C 180,E1 -4634.733,E2 -4634.733} C_VEL
LIN {X 0,Y 524.151,Z 290.093,A -85,B 0,C 180,E1 -4636.913,E2 -4636.913} C_VEL
LIN {X 0,Y 525.956,Z 300.256,A -85,B 0,C 180,E1 -4637.113,E2 -4637.113} C_VEL
LIN {X 0,Y 525.475,Z 396.911,A -85,B 0,C 180,E1 -4638.482,E2 -4638.482} C_VEL
LIN {X 0,Y 525.33,Z 410.389,A -85,B 0,C 180,E1 -4638.836,E2 -4638.836} C_VEL
LIN {X 0,Y 525.073,Z 422.887,A -85,B 0,C 180,E1 -4639.322,E2 -4639.322} C_VEL
LIN {X 0,Y 524.86,Z 433.997,A -85,B 0,C 180,E1 -4639.906,E2 -4639.906} C_VEL
LIN {X 0,Y 524.564,Z 444.46,A -85,B 0,C 180,E1 -4640.601,E2 -4640.601} C_VEL
LIN {X 0,Y 524.322,Z 454.684,A -85,B 0,C 180,E1 -4641.444,E2 -4641.444} C_VEL
LIN {X 0,Y 524.102,Z 464.661,A -85,B 0,C 180,E1 -4642.459,E2 -4642.459} C_VEL
LIN {X 0,Y 523.861,Z 473.586,A -85,B 0,C 180,E1 -4643.595,E2 -4643.595} C_VEL
LIN {X 0,Y 523.647,Z 480.913,A -85,B 0,C 180,E1 -4644.753,E2 -4644.753} C_VEL
LIN {X 0,Y 523.546,Z 487.349,A -85,B 0,C 180,E1 -4646.037,E2 -4646.037} C_VEL
LIN {X 0,Y 523.432,Z 491.391,A -85,B 0,C 180,E1 -4647.059,E2 -4647.059} C_VEL
LIN {X 0,Y 523.417,Z 495.516,A -85,B 0,C 180,E1 -4648.423,E2 -4648.423} C_VEL
LIN {X 0,Y 523.337,Z 497.413,A -85,B 0,C 180,E1 -4649.316,E2 -4649.316} C_VEL
LIN {X 0,Y 523.298,Z 499.427,A -85,B 0,C 180,E1 -4650.792,E2 -4650.792} C_VEL
LIN {X 0,Y 523.256,Z 499.891,A -85,B 0,C 180,E1 -4652.419,E2 -4652.419} C_VEL
LIN {X 0,Y 523.312,Z 498.527,A -85,B 0,C 180,E1 -4654.117,E2 -4654.117} C_VEL
LIN {X 0,Y 523.356,Z 496.188,A -85,B 0,C 180,E1 -4655.4,E2 -4655.4} C_VEL
LIN {X 0,Y 523.476,Z 492.702,A -85,B 0,C 180,E1 -4656.669,E2 -4656.669} C_VEL
LIN {X 0,Y 523.519,Z 488.022,A -85,B 0,C 180,E1 -4657.921,E2 -4657.921} C_VEL
LIN {X 0,Y 523.638,Z 481.955,A -85,B 0,C 180,E1 -4659.166,E2 -4659.166} C_VEL
LIN {X 0,Y 523.858,Z 474.323,A -85,B 0,C 180,E1 -4660.404,E2 -4660.404} C_VEL
LIN {X 0,Y 524.029,Z 466.518,A -85,B 0,C 180,E1 -4661.427,E2 -4661.427} C_VEL
LIN {X 0,Y 524.326,Z 456.624,A -85,B 0,C 180,E1 -4662.48,E2 -4662.48} C_VEL
LIN {X 0,Y 524.568,Z 446.303,A -85,B 0,C 180,E1 -4663.359,E2 -4663.359} C_VEL
LIN {X 0,Y 524.84,Z 436.012,A -85,B 0,C 180,E1 -4664.068,E2 -4664.068} C_VEL
LIN {X 0,Y 525.049,Z 425.397,A -85,B 0,C 180,E1 -4664.652,E2 -4664.652} C_VEL
LIN {X 0,Y 525.238,Z 412.663,A -85,B 0,C 180,E1 -4665.184,E2 -4665.184} C_VEL
LIN {X 0,Y 525.406,Z 399.658,A -85,B 0,C 180,E1 -4665.549,E2 -4665.549} C_VEL
LIN {X 0,Y 525.515,Z 380.923,A -85,B 0,C 180,E1 -4665.849,E2 -4665.849} C_VEL
LIN {X 0,Y 525.972,Z 299.751,A -85,B 0,C 180,E1 -4666.989,E2 -4666.989} C_VEL
LIN {X 0,Y 524.099,Z 289.491,A -85,B 0,C 180,E1 -4667.202,E2 -4667.202} C_VEL
LIN {X 0,Y 523.938,Z 275.223,A -85,B 0,C 180,E1 -4669.519,E2 -4669.519} C_VEL
LIN {X 0,Y 523.968,Z 275.217,A -85,B 0,C 180,E1 -4672.292,E2 -4672.292} C_VEL
LIN {X 0,Y 524.038,Z 275.212,A -85,B 0,C 180,E1 -4674.614,E2 -4674.614} C_VEL
LIN {X 0,Y 524.048,Z 275.205,A -85,B 0,C 180,E1 -4677.695,E2 -4677.695} C_VEL
LIN {X 0,Y 524.069,Z 275.207,A -85,B 0,C 180,E1 -4680.769,E2 -4680.769} C_VEL
LIN {X 0,Y 524.021,Z 275.214,A -85,B 0,C 180,E1 -4683.076,E2 -4683.076} C_VEL
LIN {X 0,Y 523.987,Z 275.211,A -85,B 0,C 180,E1 -4686.16,E2 -4686.16} C_VEL
LIN {X 0,Y 523.951,Z 275.22,A -85,B 0,C 180,E1 -4689.263,E2 -4689.263} C_VEL
LIN {X 0,Y 523.966,Z 275.213,A -85,B 0,C 180,E1 -4691.753,E2 -4691.753} C_VEL
LIN {X 0,Y 523.949,Z 275.222,A -85,B 0,C 180,E1 -4695.06,E2 -4695.06} C_VEL
LIN {X 0,Y 523.909,Z 275.218,A -85,B 0,C 180,E1 -4697.971,E2 -4697.971} C_VEL
LIN {X 0,Y 523.918,Z 275.218,A -85,B 0,C 180,E1 -4700.413,E2 -4700.413} C_VEL
LIN {X 0,Y 523.863,Z 275.231,A -85,B 0,C 180,E1 -4702.896,E2 -4702.896} C_VEL
LIN {X 0,Y 523.906,Z 275.223,A -85,B 0,C 180,E1 -4705.421,E2 -4705.421} C_VEL
LIN {X 0,Y 523.922,Z 275.218,A -85,B 0,C 180,E1 -4708.002,E2 -4708.002} C_VEL
LIN {X 0,Y 523.9,Z 275.226,A -85,B 0,C 180,E1 -4710.858,E2 -4710.858} C_VEL
LIN {X 0,Y 523.919,Z 275.219,A -85,B 0,C 180,E1 -4713.739,E2 -4713.739} C_VEL
LIN {X 0,Y 523.879,Z 275.224,A -85,B 0,C 180,E1 -4716.408,E2 -4716.408} C_VEL
LIN {X 0,Y 523.921,Z 275.226,A -85,B 0,C 180,E1 -4719.085,E2 -4719.085} C_VEL
LIN {X 0,Y 523.929,Z 275.216,A -85,B 0,C 180,E1 -4722.122,E2 -4722.122} C_VEL
LIN {X 0,Y 523.923,Z 275.227,A -85,B 0,C 180,E1 -4725.313,E2 -4725.313} C_VEL
LIN {X 0,Y 523.933,Z 275.219,A -85,B 0,C 180,E1 -4728.693,E2 -4728.693} C_VEL
LIN {X 0,Y 523.891,Z 275.228,A -85,B 0,C 180,E1 -4731.085,E2 -4731.085} C_VEL
LIN {X 0,Y 523.877,Z 275.228,A -85,B 0,C 180,E1 -4733.829,E2 -4733.829} C_VEL
LIN {X 0,Y 523.921,Z 275.222,A -85,B 0,C 180,E1 -4736.639,E2 -4736.639} C_VEL
LIN {X 0,Y 523.939,Z 275.228,A -85,B 0,C 180,E1 -4739.359,E2 -4739.359} C_VEL
LIN {X 0,Y 523.934,Z 275.219,A -85,B 0,C 180,E1 -4742.291,E2 -4742.291} C_VEL
LIN {X 0,Y 524.009,Z 275.239,A -85,B 0,C 180,E1 -4745.013,E2 -4745.013} C_VEL
LIN {X 0,Y 525.176,Z 282.85,A -85,B 0,C 180,E1 -4746.139,E2 -4746.139} C_VEL
LIN {X 0,Y 524.956,Z 300.259,A -85,B 0,C 180,E1 -4748.607,E2 -4748.607} C_VEL
LIN {X 0,Y 524.607,Z 322.028,A -85,B 0,C 180,E1 -4751.694,E2 -4751.694} C_VEL
LIN {X 0,Y 524.32,Z 341.665,A -85,B 0,C 180,E1 -4754.453,E2 -4754.453} C_VEL
LIN {X 0,Y 524.301,Z 344.607,A -85,B 0,C 180,E1 -4754.845,E2 -4754.845} C_VEL
LIN {X 0,Y 525.867,Z 357.419,A -85,B 0,C 180,E1 -4755.076,E2 -4755.076} C_VEL
LIN {X 0,Y 525.412,Z 454.189,A -85,B 0,C 180,E1 -4756.44,E2 -4756.44} C_VEL
LIN {X 0,Y 525.159,Z 468.009,A -85,B 0,C 180,E1 -4756.803,E2 -4756.803} C_VEL
LIN {X 0,Y 524.934,Z 480.447,A -85,B 0,C 180,E1 -4757.289,E2 -4757.289} C_VEL
LIN {X 0,Y 524.681,Z 493.052,A -85,B 0,C 180,E1 -4757.963,E2 -4757.963} C_VEL
LIN {X 0,Y 524.424,Z 503.867,A -85,B 0,C 180,E1 -4758.7,E2 -4758.7} C_VEL
LIN {X 0,Y 524.158,Z 514.229,A -85,B 0,C 180,E1 -4759.574,E2 -4759.574} C_VEL
LIN {X 0,Y 523.902,Z 523.53,A -85,B 0,C 180,E1 -4760.544,E2 -4760.544} C_VEL
LIN {X 0,Y 523.702,Z 532.581,A -85,B 0,C 180,E1 -4761.707,E2 -4761.707} C_VEL
LIN {X 0,Y 523.571,Z 539.875,A -85,B 0,C 180,E1 -4762.869,E2 -4762.869} C_VEL
LIN {X 0,Y 523.475,Z 544.788,A -85,B 0,C 180,E1 -4763.836,E2 -4763.836} C_VEL
LIN {X 0,Y 523.383,Z 549.565,A -85,B 0,C 180,E1 -4764.994,E2 -4764.994} C_VEL
LIN {X 0,Y 523.443,Z 553.221,A -85,B 0,C 180,E1 -4766.152,E2 -4766.152} C_VEL
LIN {X 0,Y 523.367,Z 555.104,A -85,B 0,C 180,E1 -4766.922,E2 -4766.922} C_VEL
LIN {X 0,Y 523.334,Z 556.515,A -85,B 0,C 180,E1 -4767.693,E2 -4767.693} C_VEL
LIN {X 0,Y 523.257,Z 558.135,A -85,B 0,C 180,E1 -4769.232,E2 -4769.232} C_VEL
LIN {X 0,Y 523.258,Z 558.357,A -85,B 0,C 180,E1 -4770.001,E2 -4770.001} C_VEL
LIN {X 0,Y 523.274,Z 557.531,A -85,B 0,C 180,E1 -4771.54,E2 -4771.54} C_VEL
LIN {X 0,Y 523.335,Z 556.533,A -85,B 0,C 180,E1 -4772.31,E2 -4772.31} C_VEL
LIN {X 0,Y 523.368,Z 555.128,A -85,B 0,C 180,E1 -4773.08,E2 -4773.08} C_VEL
LIN {X 0,Y 523.425,Z 552.171,A -85,B 0,C 180,E1 -4774.236,E2 -4774.236} C_VEL
LIN {X 0,Y 523.461,Z 548.164,A -85,B 0,C 180,E1 -4775.393,E2 -4775.393} C_VEL
LIN {X 0,Y 523.518,Z 542.893,A -85,B 0,C 180,E1 -4776.575,E2 -4776.575} C_VEL
LIN {X 0,Y 523.618,Z 536.502,A -85,B 0,C 180,E1 -4777.714,E2 -4777.714} C_VEL
LIN {X 0,Y 523.817,Z 528.401,A -85,B 0,C 180,E1 -4778.876,E2 -4778.876} C_VEL
LIN {X 0,Y 524.002,Z 520.138,A -85,B 0,C 180,E1 -4779.847,E2 -4779.847} C_VEL
LIN {X 0,Y 524.252,Z 510.058,A -85,B 0,C 180,E1 -4780.818,E2 -4780.818} C_VEL
LIN {X 0,Y 524.574,Z 498.639,A -85,B 0,C 180,E1 -4781.692,E2 -4781.692} C_VEL
LIN {X 0,Y 524.837,Z 487.473,A -85,B 0,C 180,E1 -4782.372,E2 -4782.372} C_VEL
LIN {X 0,Y 525.06,Z 475.034,A -85,B 0,C 180,E1 -4782.956,E2 -4782.956} C_VEL
